LIN {X 0,Y 304.468,Z 656.126,A -85,B 0,C 180,E1 -16142.067,E2 -16142.067} C_VEL
LIN {X 0,Y 304.044,Z 658.272,A -85,B 0,C 180,E1 -16143.694,E2 -16143.694} C_VEL
LIN {X 0,Y 303.714,Z 660.484,A -85,B 0,C 180,E1 -16145.912,E2 -16145.912} C_VEL
LIN {X 0,Y 303.547,Z 662.089,A -85,B 0,C 180,E1 -16148.692,E2 -16148.692} C_VEL
LIN {X 0,Y 303.552,Z 662.479,A -85,B 0,C 180,E1 -16150.411,E2 -16150.411} C_VEL
LIN {X 0,Y 303.63,Z 662.376,A -85,B 0,C 180,E1 -16152.209,E2 -16152.209} C_VEL
LIN {X 0,Y 303.809,Z 661.626,A -85,B 0,C 180,E1 -16154.182,E2 -16154.182} C_VEL
LIN {X 0,Y 304.102,Z 660.328,A -85,B 0,C 180,E1 -16156.106,E2 -16156.106} C_VEL
LIN {X 0,Y 304.595,Z 658.473,A -85,B 0,C 180,E1 -16158,E2 -16158} C_VEL
LIN {X 0,Y 305.42,Z 654.743,A -85,B 0,C 180,E1 -16160.682,E2 -16160.682} C_VEL
LIN {X 0,Y 306.67,Z 649.557,A -85,B 0,C 180,E1 -16163.426,E2 -16163.426} C_VEL
LIN {X 0,Y 308.375,Z 642.973,A -85,B 0,C 180,E1 -16166.107,E2 -16166.107} C_VEL
LIN {X 0,Y 310.419,Z 635.217,A -85,B 0,C 180,E1 -16168.618,E2 -16168.618} C_VEL
LIN {X 0,Y 312.569,Z 627.022,A -85,B 0,C 180,E1 -16170.788,E2 -16170.788} C_VEL
LIN {X 0,Y 315.085,Z 617.352,A -85,B 0,C 180,E1 -16172.91,E2 -16172.91} C_VEL
LIN {X 0,Y 317.539,Z 607.207,A -85,B 0,C 180,E1 -16174.766,E2 -16174.766} C_VEL
LIN {X 0,Y 320.243,Z 595.361,A -85,B 0,C 180,E1 -16176.561,E2 -16176.561} C_VEL
LIN {X 0,Y 322.857,Z 582.894,A -85,B 0,C 180,E1 -16178.112,E2 -16178.112} C_VEL
LIN {X 0,Y 325.28,Z 569.513,A -85,B 0,C 180,E1 -16179.477,E2 -16179.477} C_VEL
LIN {X 0,Y 325.963,Z 565.676,A -85,B 0,C 180,E1 -16179.818,E2 -16179.818} C_VEL
LIN {X 0,Y 325.947,Z 562.448,A -85,B 0,C 180,E1 -16180.17,E2 -16180.17} C_VEL
LIN {X 0,Y 324.622,Z 558.931,A -85,B 0,C 180,E1 -16180.704,E2 -16180.704} C_VEL
LIN {X 0,Y 321.402,Z 554.854,A -85,B 0,C 180,E1 -16181.521,E2 -16181.521} C_VEL
LIN {X 0,Y 315.876,Z 549.196,A -85,B 0,C 180,E1 -16182.776,E2 -16182.776} C_VEL
LIN {X 0,Y 313.449,Z 544.969,A -85,B 0,C 180,E1 -16183.488,E2 -16183.488} C_VEL
LIN {X 0,Y 308.452,Z 533.574,A -85,B 0,C 180,E1 -16185.105,E2 -16185.105} C_VEL
LIN {X 0,Y 303.295,Z 523.807,A -85,B 0,C 180,E1 -16186.575,E2 -16186.575} C_VEL
LIN {X 0,Y 300.999,Z 519.913,A -85,B 0,C 180,E1 -16187.184,E2 -16187.184} C_VEL
LIN {X 0,Y 299.322,Z 517.279,A -85,B 0,C 180,E1 -16187.628,E2 -16187.628} C_VEL
LIN {X 0,Y 298.927,Z 515.725,A -85,B 0,C 180,E1 -16187.783,E2 -16187.783} C_VEL
LIN {X 0,Y 299.077,Z 513.977,A -85,B 0,C 180,E1 -16191.894,E2 -16191.894} C_VEL
LIN {X 0,Y 298.86,Z 513.035,A -85,B 0,C 180,E1 -16194.602,E2 -16194.602} C_VEL
LIN {X 0,Y 298.922,Z 511.875,A -85,B 0,C 180,E1 -16198.652,E2 -16198.652} C_VEL
LIN {X 0,Y 298.922,Z 511.874,A -85,B 0,C 180,E1 -16201.347,E2 -16201.347} C_VEL
LIN {X 0,Y 298.796,Z 511.89,A -85,B 0,C 180,E1 -16206.753,E2 -16206.753} C_VEL
LIN {X 0,Y 298.679,Z 511.903,A -85,B 0,C 180,E1 -16209.48,E2 -16209.48} C_VEL
LIN {X 0,Y 298.55,Z 511.918,A -85,B 0,C 180,E1 -16213.615,E2 -16213.615} C_VEL
LIN {X 0,Y 298.546,Z 511.923,A -85,B 0,C 180,E1 -16216.408,E2 -16216.408} C_VEL
LIN {X 0,Y 298.509,Z 511.924,A -85,B 0,C 180,E1 -16219.654,E2 -16219.654} C_VEL
LIN {X 0,Y 298.446,Z 512.07,A -85,B 0,C 180,E1 -16222.134,E2 -16222.134} C_VEL
LIN {X 0,Y 298.697,Z 513.171,A -85,B 0,C 180,E1 -16225.056,E2 -16225.056} C_VEL
LIN {X 0,Y 298.927,Z 514.632,A -85,B 0,C 180,E1 -16228.048,E2 -16228.048} C_VEL
LIN {X 0,Y 299.194,Z 516.442,A -85,B 0,C 180,E1 -16231.116,E2 -16231.116} C_VEL
LIN {X 0,Y 299.664,Z 519.004,A -85,B 0,C 180,E1 -16234.83,E2 -16234.83} C_VEL
LIN {X 0,Y 300.312,Z 522.622,A -85,B 0,C 180,E1 -16239.187,E2 -16239.187} C_VEL
LIN {X 0,Y 300.797,Z 525.954,A -85,B 0,C 180,E1 -16242.654,E2 -16242.654} C_VEL
LIN {X 0,Y 301.367,Z 529.88,A -85,B 0,C 180,E1 -16246.297,E2 -16246.297} C_VEL
LIN {X 0,Y 301.234,Z 532.28,A -85,B 0,C 180,E1 -16248.295,E2 -16248.295} C_VEL
LIN {X 0,Y 300.435,Z 537.264,A -85,B 0,C 180,E1 -16252.116,E2 -16252.116} C_VEL
LIN {X 0,Y 300.324,Z 537.751,A -85,B 0,C 180,E1 -16252.464,E2 -16252.464} C_VEL
LIN {X 0,Y 301.249,Z 540.977,A -85,B 0,C 180,E1 -16252.761,E2 -16252.761} C_VEL
LIN {X 0,Y 302.452,Z 543.428,A -85,B 0,C 180,E1 -16253.081,E2 -16253.081} C_VEL
LIN {X 0,Y 307.21,Z 556.096,A -85,B 0,C 180,E1 -16254.515,E2 -16254.515} C_VEL
LIN {X 0,Y 310.981,Z 569.368,A -85,B 0,C 180,E1 -16255.971,E2 -16255.971} C_VEL
LIN {X 0,Y 313.752,Z 583.061,A -85,B 0,C 180,E1 -16257.48,E2 -16257.48} C_VEL
LIN {X 0,Y 315.221,Z 596.358,A -85,B 0,C 180,E1 -16258.972,E2 -16258.972} C_VEL
LIN {X 0,Y 315.648,Z 607.148,A -85,B 0,C 180,E1 -16260.266,E2 -16260.266} C_VEL
LIN {X 0,Y 314.902,Z 611.825,A -85,B 0,C 180,E1 -16260.777,E2 -16260.777} C_VEL
LIN {X 0,Y 311.977,Z 624.765,A -85,B 0,C 180,E1 -16262.314,E2 -16262.314} C_VEL
LIN {X 0,Y 309.129,Z 636.736,A -85,B 0,C 180,E1 -16264.046,E2 -16264.046} C_VEL
LIN {X 0,Y 306.332,Z 647.818,A -85,B 0,C 180,E1 -16265.969,E2 -16265.969} C_VEL
LIN {X 0,Y 303.981,Z 657.256,A -85,B 0,C 180,E1 -16267.935,E2 -16267.935} C_VEL
LIN {X 0,Y 301.707,Z 666.564,A -85,B 0,C 180,E1 -16270.259,E2 -16270.259} C_VEL
LIN {X 0,Y 299.707,Z 675.414,A -85,B 0,C 180,E1 -16272.955,E2 -16272.955} C_VEL
LIN {X 0,Y 298.197,Z 682.598,A -85,B 0,C 180,E1 -16275.672,E2 -16275.672} C_VEL
LIN {X 0,Y 297.264,Z 688.305,A -85,B 0,C 180,E1 -16278.406,E2 -16278.406} C_VEL
LIN {X 0,Y 296.881,Z 691.721,A -85,B 0,C 180,E1 -16280.461,E2 -16280.461} C_VEL
LIN {X 0,Y 296.637,Z 695.166,A -85,B 0,C 180,E1 -16283.196,E2 -16283.196} C_VEL
LIN {X 0,Y 296.651,Z 697.347,A -85,B 0,C 180,E1 -16285.924,E2 -16285.924} C_VEL
LIN {X 0,Y 296.763,Z 698.349,A -85,B 0,C 180,E1 -16288.642,E2 -16288.642} C_VEL
LIN {X 0,Y 296.887,Z 698.412,A -85,B 0,C 180,E1 -16289.999,E2 -16289.999} C_VEL
LIN {X 0,Y 296.672,Z 697.618,A -85,B 0,C 180,E1 -16292.715,E2 -16292.715} C_VEL
LIN {X 0,Y 296.689,Z 695.633,A -85,B 0,C 180,E1 -16295.436,E2 -16295.436} C_VEL
LIN {X 0,Y 296.777,Z 692.368,A -85,B 0,C 180,E1 -16298.168,E2 -16298.168} C_VEL
LIN {X 0,Y 297.068,Z 687.756,A -85,B 0,C 180,E1 -16300.909,E2 -16300.909} C_VEL
LIN {X 0,Y 297.844,Z 681.725,A -85,B 0,C 180,E1 -16303.647,E2 -16303.647} C_VEL
LIN {X 0,Y 299.149,Z 674.123,A -85,B 0,C 180,E1 -16306.374,E2 -16306.374} C_VEL
LIN {X 0,Y 300.619,Z 665.958,A -85,B 0,C 180,E1 -16308.75,E2 -16308.75} C_VEL
LIN {X 0,Y 302.441,Z 657.688,A -85,B 0,C 180,E1 -16310.754,E2 -16310.754} C_VEL
LIN {X 0,Y 304.456,Z 647.468,A -85,B 0,C 180,E1 -16312.846,E2 -16312.846} C_VEL
LIN {X 0,Y 306.936,Z 635.389,A -85,B 0,C 180,E1 -16314.88,E2 -16314.88} C_VEL
LIN {X 0,Y 309.172,Z 623.827,A -85,B 0,C 180,E1 -16316.493,E2 -16316.493} C_VEL
LIN {X 0,Y 311.592,Z 611.493,A -85,B 0,C 180,E1 -16317.905,E2 -16317.905} C_VEL
LIN {X 0,Y 312.384,Z 605.5,A -85,B 0,C 180,E1 -16318.519,E2 -16318.519} C_VEL
LIN {X 0,Y 310.846,Z 591.329,A -85,B 0,C 180,E1 -16320.03,E2 -16320.03} C_VEL
LIN {X 0,Y 308.538,Z 577.479,A -85,B 0,C 180,E1 -16321.332,E2 -16321.332} C_VEL
LIN {X 0,Y 305.347,Z 563.007,A -85,B 0,C 180,E1 -16322.536,E2 -16322.536} C_VEL
LIN {X 0,Y 301.249,Z 548.178,A -85,B 0,C 180,E1 -16323.625,E2 -16323.625} C_VEL
LIN {X 0,Y 299.596,Z 542.829,A -85,B 0,C 180,E1 -16323.986,E2 -16323.986} C_VEL
LIN {X 0,Y 299.525,Z 541.899,A -85,B 0,C 180,E1 -16324.059,E2 -16324.059} C_VEL
LIN {X 0,Y 300.214,Z 536.845,A -85,B 0,C 180,E1 -16327.491,E2 -16327.491} C_VEL
LIN {X 0,Y 301.015,Z 532.092,A -85,B 0,C 180,E1 -16330.822,E2 -16330.822} C_VEL
LIN {X 0,Y 301.291,Z 529.646,A -85,B 0,C 180,E1 -16332.566,E2 -16332.566} C_VEL
LIN {X 0,Y 300.918,Z 525.827,A -85,B 0,C 180,E1 -16335.521,E2 -16335.521} C_VEL
LIN {X 0,Y 300.088,Z 521.552,A -85,B 0,C 180,E1 -16339.024,E2 -16339.024} C_VEL
LIN {X 0,Y 299.269,Z 517.042,A -85,B 0,C 180,E1 -16342.98,E2 -16342.98} C_VEL
LIN {X 0,Y 298.814,Z 514.18,A -85,B 0,C 180,E1 -16345.635,E2 -16345.635} C_VEL
LIN {X 0,Y 298.394,Z 511.938,A -85,B 0,C 180,E1 -16347.981,E2 -16347.981} C_VEL
LIN {X 0,Y 298.461,Z 511.933,A -85,B 0,C 180,E1 -16351.905,E2 -16351.905} C_VEL
LIN {X 0,Y 298.475,Z 511.93,A -85,B 0,C 180,E1 -16354.924,E2 -16354.924} C_VEL
LIN {X 0,Y 298.431,Z 511.938,A -85,B 0,C 180,E1 -16359.314,E2 -16359.314} C_VEL
LIN {X 0,Y 298.529,Z 511.923,A -85,B 0,C 180,E1 -16362.179,E2 -16362.179} C_VEL
LIN {X 0,Y 298.585,Z 511.916,A -85,B 0,C 180,E1 -16364.995,E2 -16364.995} C_VEL
LIN {X 0,Y 298.587,Z 511.914,A -85,B 0,C 180,E1 -16369.147,E2 -16369.147} C_VEL
LIN {X 0,Y 298.75,Z 511.891,A -85,B 0,C 180,E1 -16371.886,E2 -16371.886} C_VEL
LIN {X 0,Y 298.654,Z 511.905,A -85,B 0,C 180,E1 -16374.599,E2 -16374.599} C_VEL
LIN {X 0,Y 298.919,Z 511.869,A -85,B 0,C 180,E1 -16378.653,E2 -16378.653} C_VEL
LIN {X 0,Y 298.917,Z 511.865,A -85,B 0,C 180,E1 -16381.348,E2 -16381.348} C_VEL
LIN {X 0,Y 298.782,Z 511.89,A -85,B 0,C 180,E1 -16386.755,E2 -16386.755} C_VEL
LIN {X 0,Y 298.627,Z 511.908,A -85,B 0,C 180,E1 -16389.483,E2 -16389.483} C_VEL
LIN {X 0,Y 298.544,Z 511.913,A -85,B 0,C 180,E1 -16393.616,E2 -16393.616} C_VEL
LIN {X 0,Y 298.541,Z 511.919,A -85,B 0,C 180,E1 -16396.41,E2 -16396.41} C_VEL
LIN {X 0,Y 298.504,Z 511.926,A -85,B 0,C 180,E1 -16399.656,E2 -16399.656} C_VEL
LIN {X 0,Y 298.451,Z 511.922,A -85,B 0,C 180,E1 -16403.599,E2 -16403.599} C_VEL
LIN {X 0,Y 298.484,Z 511.922,A -85,B 0,C 180,E1 -16406.576,E2 -16406.576} C_VEL
LIN {X 0,Y 298.417,Z 511.94,A -85,B 0,C 180,E1 -16409.642,E2 -16409.642} C_VEL
LIN {X 0,Y 298.393,Z 511.936,A -85,B 0,C 180,E1 -16412.801,E2 -16412.801} C_VEL
LIN {X 0,Y 298.467,Z 511.92,A -85,B 0,C 180,E1 -16416.815,E2 -16416.815} C_VEL
LIN {X 0,Y 298.454,Z 511.933,A -85,B 0,C 180,E1 -16421.251,E2 -16421.251} C_VEL
LIN {X 0,Y 298.487,Z 511.923,A -85,B 0,C 180,E1 -16425.062,E2 -16425.062} C_VEL
LIN {X 0,Y 298.455,Z 511.929,A -85,B 0,C 180,E1 -16428.898,E2 -16428.898} C_VEL
LIN {X 0,Y 298.469,Z 511.931,A -85,B 0,C 180,E1 -16433.188,E2 -16433.188} C_VEL
LIN {X 0,Y 298.395,Z 511.936,A -85,B 0,C 180,E1 -16437.201,E2 -16437.201} C_VEL
LIN {X 0,Y 298.433,Z 511.935,A -85,B 0,C 180,E1 -16440.616,E2 -16440.616} C_VEL
LIN {X 0,Y 298.485,Z 511.925,A -85,B 0,C 180,E1 -16443.475,E2 -16443.475} C_VEL
LIN {X 0,Y 298.438,Z 511.933,A -85,B 0,C 180,E1 -16446.698,E2 -16446.698} C_VEL
LIN {X 0,Y 298.542,Z 511.916,A -85,B 0,C 180,E1 -16450.758,E2 -16450.758} C_VEL
LIN {X 0,Y 298.597,Z 511.912,A -85,B 0,C 180,E1 -16454.996,E2 -16454.996} C_VEL
LIN {X 0,Y 298.595,Z 511.915,A -85,B 0,C 180,E1 -16459.148,E2 -16459.148} C_VEL
LIN {X 0,Y 298.723,Z 511.901,A -85,B 0,C 180,E1 -16461.886,E2 -16461.886} C_VEL
LIN {X 0,Y 298.66,Z 511.903,A -85,B 0,C 180,E1 -16464.6,E2 -16464.6} C_VEL
LIN {X 0,Y 298.929,Z 511.872,A -85,B 0,C 180,E1 -16468.654,E2 -16468.654} C_VEL
LIN {X 0,Y 298.863,Z 511.881,A -85,B 0,C 180,E1 -16471.348,E2 -16471.348} C_VEL
LIN {X 0,Y 298.253,Z 512.084,A -85,B 0,C 180,E1 -16476.003,E2 -16476.003} C_VEL
LIN {X 0,Y 299.348,Z 515.022,A -85,B 0,C 180,E1 -16476.234,E2 -16476.234} C_VEL
LIN {X 0,Y 302.643,Z 522.4,A -85,B 0,C 180,E1 -16476.899,E2 -16476.899} C_VEL
LIN {X 0,Y 307.781,Z 536.221,A -85,B 0,C 180,E1 -16478.189,E2 -16478.189} C_VEL
LIN {X 0,Y 311.731,Z 548.462,A -85,B 0,C 180,E1 -16479.446,E2 -16479.446} C_VEL
LIN {X 0,Y 315.162,Z 561.803,A -85,B 0,C 180,E1 -16480.942,E2 -16480.942} C_VEL
LIN {X 0,Y 313.165,Z 576.214,A -85,B 0,C 180,E1 -16482.31,E2 -16482.31} C_VEL
LIN {X 0,Y 310.649,Z 590.58,A -85,B 0,C 180,E1 -16484.004,E2 -16484.004} C_VEL
LIN {X 0,Y 308.481,Z 602.271,A -85,B 0,C 180,E1 -16485.697,E2 -16485.697} C_VEL
LIN {X 0,Y 306.015,Z 613.873,A -85,B 0,C 180,E1 -16487.717,E2 -16487.717} C_VEL
LIN {X 0,Y 303.761,Z 624.438,A -85,B 0,C 180,E1 -16489.959,E2 -16489.959} C_VEL
LIN {X 0,Y 301.856,Z 633.291,A -85,B 0,C 180,E1 -16492.231,E2 -16492.231} C_VEL
LIN {X 0,Y 300.067,Z 641.854,A -85,B 0,C 180,E1 -16494.935,E2 -16494.935} C_VEL
LIN {X 0,Y 298.855,Z 648.075,A -85,B 0,C 180,E1 -16497.369,E2 -16497.369} C_VEL
LIN {X 0,Y 298.014,Z 652.821,A -85,B 0,C 180,E1 -16499.686,E2 -16499.686} C_VEL
LIN {X 0,Y 297.458,Z 656.235,A -85,B 0,C 180,E1 -16501.725,E2 -16501.725} C_VEL
LIN {X 0,Y 296.798,Z 659.814,A -85,B 0,C 180,E1 -16504.632,E2 -16504.632} C_VEL
LIN {X 0,Y 296.598,Z 661.257,A -85,B 0,C 180,E1 -16506.326,E2 -16506.326} C_VEL
LIN {X 0,Y 296.475,Z 662.439,A -85,B 0,C 180,E1 -16508.53,E2 -16508.53} C_VEL
LIN {X 0,Y 296.478,Z 662.939,A -85,B 0,C 180,E1 -16510.662,E2 -16510.662} C_VEL
LIN {X 0,Y 296.636,Z 662.495,A -85,B 0,C 180,E1 -16513.399,E2 -16513.399} C_VEL
LIN {X 0,Y 296.868,Z 661.589,A -85,B 0,C 180,E1 -16515.252,E2 -16515.252} C_VEL
LIN {X 0,Y 297.275,Z 660.07,A -85,B 0,C 180,E1 -16517.129,E2 -16517.129} C_VEL
LIN {X 0,Y 298.067,Z 657.03,A -85,B 0,C 180,E1 -16519.775,E2 -16519.775} C_VEL
LIN {X 0,Y 299.357,Z 651.736,A -85,B 0,C 180,E1 -16522.96,E2 -16522.96} C_VEL
LIN {X 0,Y 300.826,Z 646.331,A -85,B 0,C 180,E1 -16525.443,E2 -16525.443} C_VEL
LIN {X 0,Y 302.83,Z 639.188,A -85,B 0,C 180,E1 -16528.043,E2 -16528.043} C_VEL
LIN {X 0,Y 305.305,Z 630.25,A -85,B 0,C 180,E1 -16530.648,E2 -16530.648} C_VEL
LIN {X 0,Y 307.914,Z 620.784,A -85,B 0,C 180,E1 -16532.892,E2 -16532.892} C_VEL
LIN {X 0,Y 310.755,Z 609.932,A -85,B 0,C 180,E1 -16535.007,E2 -16535.007} C_VEL
LIN {X 0,Y 313.475,Z 598.769,A -85,B 0,C 180,E1 -16536.809,E2 -16536.809} C_VEL
LIN {X 0,Y 316.378,Z 585.853,A -85,B 0,C 180,E1 -16538.517,E2 -16538.517} C_VEL
LIN {X 0,Y 318.946,Z 572.612,A -85,B 0,C 180,E1 -16539.944,E2 -16539.944} C_VEL
LIN {X 0,Y 319.911,Z 567.296,A -85,B 0,C 180,E1 -16540.426,E2 -16540.426} C_VEL
LIN {X 0,Y 317.233,Z 556.251,A -85,B 0,C 180,E1 -16541.931,E2 -16541.931} C_VEL
LIN {X 0,Y 313.449,Z 544.969,A -85,B 0,C 180,E1 -16543.488,E2 -16543.488} C_VEL
LIN {X 0,Y 311.819,Z 542.414,A -85,B 0,C 180,E1 -16543.954,E2 -16543.954} C_VEL
LIN {X 0,Y 307.83,Z 539.626,A -85,B 0,C 180,E1 -16544.814,E2 -16544.814} C_VEL
LIN {X 0,Y 303.71,Z 536.917,A -85,B 0,C 180,E1 -16545.693,E2 -16545.693} C_VEL
LIN {X 0,Y 301.871,Z 534.458,A -85,B 0,C 180,E1 -16546.182,E2 -16546.182} C_VEL
LIN {X 0,Y 298.564,Z 528.116,A -85,B 0,C 180,E1 -16547.207,E2 -16547.207} C_VEL
LIN {X 0,Y 296.802,Z 524.957,A -85,B 0,C 180,E1 -16547.738,E2 -16547.738} C_VEL
LIN {X 0,Y 294.822,Z 521.445,A -85,B 0,C 180,E1 -16548.31,E2 -16548.31} C_VEL
LIN {X 0,Y 292.662,Z 518.54,A -85,B 0,C 180,E1 -16548.894,E2 -16548.894} C_VEL
LIN {X 0,Y 291.963,Z 516.396,A -85,B 0,C 180,E1 -16549.16,E2 -16549.16} C_VEL
LIN {X 0,Y 292.098,Z 515.364,A -85,B 0,C 180,E1 -16551.699,E2 -16551.699} C_VEL
LIN {X 0,Y 291.915,Z 514.421,A -85,B 0,C 180,E1 -16554.473,E2 -16554.473} C_VEL
LIN {X 0,Y 291.946,Z 513.188,A -85,B 0,C 180,E1 -16558.62,E2 -16558.62} C_VEL
LIN {X 0,Y 291.888,Z 512.75,A -85,B 0,C 180,E1 -16561.379,E2 -16561.379} C_VEL
LIN {X 0,Y 291.745,Z 512.767,A -85,B 0,C 180,E1 -16566.917,E2 -16566.917} C_VEL
LIN {X 0,Y 291.628,Z 512.781,A -85,B 0,C 180,E1 -16569.711,E2 -16569.711} C_VEL
LIN {X 0,Y 291.52,Z 512.795,A -85,B 0,C 180,E1 -16573.95,E2 -16573.95} C_VEL
LIN {X 0,Y 291.485,Z 512.8,A -85,B 0,C 180,E1 -16576.817,E2 -16576.817} C_VEL
LIN {X 0,Y 291.482,Z 512.993,A -85,B 0,C 180,E1 -16579.892,E2 -16579.892} C_VEL
LIN {X 0,Y 291.676,Z 514.441,A -85,B 0,C 180,E1 -16584.18,E2 -16584.18} C_VEL
LIN {X 0,Y 291.943,Z 515.792,A -85,B 0,C 180,E1 -16587.218,E2 -16587.218} C_VEL
LIN {X 0,Y 292.188,Z 517.522,A -85,B 0,C 180,E1 -16590.338,E2 -16590.338} C_VEL
LIN {X 0,Y 292.534,Z 519.609,A -85,B 0,C 180,E1 -16593.543,E2 -16593.543} C_VEL
LIN {X 0,Y 292.983,Z 522.099,A -85,B 0,C 180,E1 -16596.847,E2 -16596.847} C_VEL
LIN {X 0,Y 293.498,Z 525.046,A -85,B 0,C 180,E1 -16600.28,E2 -16600.28} C_VEL
LIN {X 0,Y 294.068,Z 528.9,A -85,B 0,C 180,E1 -16604.195,E2 -16604.195} C_VEL
LIN {X 0,Y 294.367,Z 531.02,A -85,B 0,C 180,E1 -16606.182,E2 -16606.182} C_VEL
LIN {X 0,Y 294.101,Z 534.266,A -85,B 0,C 180,E1 -16608.917,E2 -16608.917} C_VEL
LIN {X 0,Y 293.625,Z 537.124,A -85,B 0,C 180,E1 -16611.157,E2 -16611.157} C_VEL
LIN {X 0,Y 294.568,Z 540.375,A -85,B 0,C 180,E1 -16611.483,E2 -16611.483} C_VEL
LIN {X 0,Y 295.873,Z 543.008,A -85,B 0,C 180,E1 -16611.86,E2 -16611.86} C_VEL
LIN {X 0,Y 301.07,Z 556.672,A -85,B 0,C 180,E1 -16613.538,E2 -16613.538} C_VEL
LIN {X 0,Y 304.668,Z 569.174,A -85,B 0,C 180,E1 -16615.01,E2 -16615.01} C_VEL
LIN {X 0,Y 307.4,Z 582.594,A -85,B 0,C 180,E1 -16616.563,E2 -16616.563} C_VEL
LIN {X 0,Y 308.824,Z 594.993,A -85,B 0,C 180,E1 -16618.015,E2 -16618.015} C_VEL
LIN {X 0,Y 309.388,Z 608.259,A -85,B 0,C 180,E1 -16619.677,E2 -16619.677} C_VEL
LIN {X 0,Y 308.086,Z 615.217,A -85,B 0,C 180,E1 -16620.468,E2 -16620.468} C_VEL
LIN {X 0,Y 304.882,Z 628.503,A -85,B 0,C 180,E1 -16622.173,E2 -16622.173} C_VEL
LIN {X 0,Y 301.721,Z 640.753,A -85,B 0,C 180,E1 -16624.103,E2 -16624.103} C_VEL
LIN {X 0,Y 298.552,Z 652.667,A -85,B 0,C 180,E1 -16626.41,E2 -16626.41} C_VEL
LIN {X 0,Y 296.015,Z 662.664,A -85,B 0,C 180,E1 -16628.773,E2 -16628.773} C_VEL
LIN {X 0,Y 293.793,Z 671.055,A -85,B 0,C 180,E1 -16631.159,E2 -16631.159} C_VEL
LIN {X 0,Y 291.966,Z 678.98,A -85,B 0,C 180,E1 -16633.929,E2 -16633.929} C_VEL
LIN {X 0,Y 290.691,Z 685.343,A -85,B 0,C 180,E1 -16636.721,E2 -16636.721} C_VEL
LIN {X 0,Y 289.91,Z 690.326,A -85,B 0,C 180,E1 -16639.524,E2 -16639.524} C_VEL
LIN {X 0,Y 289.634,Z 693.242,A -85,B 0,C 180,E1 -16641.628,E2 -16641.628} C_VEL
LIN {X 0,Y 289.554,Z 696.035,A -85,B 0,C 180,E1 -16644.428,E2 -16644.428} C_VEL
LIN {X 0,Y 289.587,Z 697.586,A -85,B 0,C 180,E1 -16647.217,E2 -16647.217} C_VEL
LIN {X 0,Y 289.798,Z 697.972,A -85,B 0,C 180,E1 -16649.999,E2 -16649.999} C_VEL
LIN {X 0,Y 289.595,Z 697.146,A -85,B 0,C 180,E1 -16652.781,E2 -16652.781} C_VEL
LIN {X 0,Y 289.622,Z 695.126,A -85,B 0,C 180,E1 -16655.569,E2 -16655.569} C_VEL
LIN {X 0,Y 289.699,Z 691.837,A -85,B 0,C 180,E1 -16658.369,E2 -16658.369} C_VEL
LIN {X 0,Y 290.028,Z 687.187,A -85,B 0,C 180,E1 -16661.177,E2 -16661.177} C_VEL
LIN {X 0,Y 290.866,Z 681.11,A -85,B 0,C 180,E1 -16663.981,E2 -16663.981} C_VEL
LIN {X 0,Y 292.251,Z 673.454,A -85,B 0,C 180,E1 -16666.772,E2 -16666.772} C_VEL
LIN {X 0,Y 293.825,Z 665.23,A -85,B 0,C 180,E1 -16669.2,E2 -16669.2} C_VEL
LIN {X 0,Y 295.673,Z 656.884,A -85,B 0,C 180,E1 -16671.252,E2 -16671.252} C_VEL
LIN {X 0,Y 297.78,Z 646.834,A -85,B 0,C 180,E1 -16673.338,E2 -16673.338} C_VEL
LIN {X 0,Y 300.4,Z 634.412,A -85,B 0,C 180,E1 -16675.459,E2 -16675.459} C_VEL
LIN {X 0,Y 303.074,Z 621.461,A -85,B 0,C 180,E1 -16677.256,E2 -16677.256} C_VEL
LIN {X 0,Y 305.564,Z 608.497,A -85,B 0,C 180,E1 -16678.716,E2 -16678.716} C_VEL
LIN {X 0,Y 305.611,Z 605.241,A -85,B 0,C 180,E1 -16679.089,E2 -16679.089} C_VEL
LIN {X 0,Y 304.02,Z 590.859,A -85,B 0,C 180,E1 -16680.673,E2 -16680.673} C_VEL
LIN {X 0,Y 301.593,Z 576.374,A -85,B 0,C 180,E1 -16682.077,E2 -16682.077} C_VEL
LIN {X 0,Y 298.299,Z 561.765,A -85,B 0,C 180,E1 -16683.324,E2 -16683.324} C_VEL
LIN {X 0,Y 294.285,Z 547.64,A -85,B 0,C 180,E1 -16684.395,E2 -16684.395} C_VEL
LIN {X 0,Y 292.687,Z 542.207,A -85,B 0,C 180,E1 -16684.77,E2 -16684.77} C_VEL
LIN {X 0,Y 292.652,Z 541.489,A -85,B 0,C 180,E1 -16684.855,E2 -16684.855} C_VEL
LIN {X 0,Y 293.586,Z 535.209,A -85,B 0,C 180,E1 -16689.276,E2 -16689.276} C_VEL
LIN {X 0,Y 294.19,Z 531.145,A -85,B 0,C 180,E1 -16692.221,E2 -16692.221} C_VEL
LIN {X 0,Y 294.167,Z 528.562,A -85,B 0,C 180,E1 -16694.215,E2 -16694.215} C_VEL
LIN {X 0,Y 293.344,Z 523.995,A -85,B 0,C 180,E1 -16697.96,E2 -16697.96} C_VEL
LIN {X 0,Y 292.383,Z 518.868,A -85,B 0,C 180,E1 -16702.485,E2 -16702.485} C_VEL
LIN {X 0,Y 291.71,Z 514.79,A -85,B 0,C 180,E1 -16706.35,E2 -16706.35} C_VEL
LIN {X 0,Y 291.341,Z 512.817,A -85,B 0,C 180,E1 -16708.354,E2 -16708.354} C_VEL
LIN {X 0,Y 291.379,Z 512.815,A -85,B 0,C 180,E1 -16711.159,E2 -16711.159} C_VEL
LIN {X 0,Y 291.408,Z 512.81,A -85,B 0,C 180,E1 -16714.272,E2 -16714.272} C_VEL
LIN {X 0,Y 291.366,Z 512.818,A -85,B 0,C 180,E1 -16717.299,E2 -16717.299} C_VEL
LIN {X 0,Y 291.45,Z 512.805,A -85,B 0,C 180,E1 -16720.27,E2 -16720.27} C_VEL
LIN {X 0,Y 291.547,Z 512.791,A -85,B 0,C 180,E1 -16724.624,E2 -16724.624} C_VEL
LIN {X 0,Y 291.53,Z 512.791,A -85,B 0,C 180,E1 -16728.881,E2 -16728.881} C_VEL
LIN {X 0,Y 291.7,Z 512.767,A -85,B 0,C 180,E1 -16731.689,E2 -16731.689} C_VEL
LIN {X 0,Y 291.624,Z 512.781,A -85,B 0,C 180,E1 -16734.469,E2 -16734.469} C_VEL
LIN {X 0,Y 291.885,Z 512.745,A -85,B 0,C 180,E1 -16738.621,E2 -16738.621} C_VEL
LIN {X 0,Y 291.883,Z 512.739,A -85,B 0,C 180,E1 -16741.38,E2 -16741.38} C_VEL
LIN {X 0,Y 291.73,Z 512.769,A -85,B 0,C 180,E1 -16746.919,E2 -16746.919} C_VEL
LIN {X 0,Y 291.567,Z 512.784,A -85,B 0,C 180,E1 -16749.715,E2 -16749.715} C_VEL
LIN {X 0,Y 291.514,Z 512.791,A -85,B 0,C 180,E1 -16753.951,E2 -16753.951} C_VEL
LIN {X 0,Y 291.48,Z 512.798,A -85,B 0,C 180,E1 -16756.819,E2 -16756.819} C_VEL
LIN {X 0,Y 291.444,Z 512.803,A -85,B 0,C 180,E1 -16759.876,E2 -16759.876} C_VEL
LIN {X 0,Y 291.394,Z 512.797,A -85,B 0,C 180,E1 -16764.206,E2 -16764.206} C_VEL
LIN {X 0,Y 291.417,Z 512.805,A -85,B 0,C 180,E1 -16767.273,E2 -16767.273} C_VEL
LIN {X 0,Y 291.334,Z 512.817,A -85,B 0,C 180,E1 -16770.438,E2 -16770.438} C_VEL
LIN {X 0,Y 291.341,Z 512.811,A -85,B 0,C 180,E1 -16773.7,E2 -16773.7} C_VEL
LIN {X 0,Y 291.401,Z 512.802,A -85,B 0,C 180,E1 -16777.263,E2 -16777.263} C_VEL
LIN {X 0,Y 291.403,Z 512.809,A -85,B 0,C 180,E1 -16780.632,E2 -16780.632} C_VEL
LIN {X 0,Y 291.404,Z 512.804,A -85,B 0,C 180,E1 -16784.381,E2 -16784.381} C_VEL
LIN {X 0,Y 291.389,Z 512.809,A -85,B 0,C 180,E1 -16788.391,E2 -16788.391} C_VEL
LIN {X 0,Y 291.387,Z 512.814,A -85,B 0,C 180,E1 -16791.166,E2 -16791.166} C_VEL
LIN {X 0,Y 291.385,Z 512.806,A -85,B 0,C 180,E1 -16794.631,E2 -16794.631} C_VEL
LIN {X 0,Y 291.372,Z 512.817,A -85,B 0,C 180,E1 -16797.952,E2 -16797.952} C_VEL
LIN {X 0,Y 291.384,Z 512.815,A -85,B 0,C 180,E1 -16801.16,E2 -16801.16} C_VEL
LIN {X 0,Y 291.419,Z 512.805,A -85,B 0,C 180,E1 -16804.273,E2 -16804.273} C_VEL
LIN {X 0,Y 291.384,Z 512.815,A -85,B 0,C 180,E1 -16807.301,E2 -16807.301} C_VEL
LIN {X 0,Y 291.461,Z 512.798,A -85,B 0,C 180,E1 -16810.271,E2 -16810.271} C_VEL
LIN {X 0,Y 291.558,Z 512.788,A -85,B 0,C 180,E1 -16814.625,E2 -16814.625} C_VEL
LIN {X 0,Y 291.539,Z 512.793,A -85,B 0,C 180,E1 -16818.882,E2 -16818.882} C_VEL
LIN {X 0,Y 291.672,Z 512.779,A -85,B 0,C 180,E1 -16821.688,E2 -16821.688} C_VEL
LIN {X 0,Y 291.63,Z 512.779,A -85,B 0,C 180,E1 -16824.469,E2 -16824.469} C_VEL
LIN {X 0,Y 291.895,Z 512.749,A -85,B 0,C 180,E1 -16828.621,E2 -16828.621} C_VEL
LIN {X 0,Y 291.821,Z 512.758,A -85,B 0,C 180,E1 -16831.381,E2 -16831.381} C_VEL
LIN {X 0,Y 291.287,Z 512.827,A -85,B 0,C 180,E1 -16835.192,E2 -16835.192} C_VEL
LIN {X 0,Y 292.436,Z 515.906,A -85,B 0,C 180,E1 -16835.474,E2 -16835.474} C_VEL
LIN {X 0,Y 296.593,Z 524.963,A -85,B 0,C 180,E1 -16836.35,E2 -16836.35} C_VEL
LIN {X 0,Y 301.963,Z 539.695,A -85,B 0,C 180,E1 -16837.805,E2 -16837.805} C_VEL
LIN {X 0,Y 306.01,Z 552.987,A -85,B 0,C 180,E1 -16839.252,E2 -16839.252} C_VEL
LIN {X 0,Y 308.645,Z 563.578,A -85,B 0,C 180,E1 -16840.496,E2 -16840.496} C_VEL
LIN {X 0,Y 306.493,Z 577.904,A -85,B 0,C 180,E1 -16841.91,E2 -16841.91} C_VEL
LIN {X 0,Y 304.021,Z 591.48,A -85,B 0,C 180,E1 -16843.565,E2 -16843.565} C_VEL
LIN {X 0,Y 301.688,Z 603.538,A -85,B 0,C 180,E1 -16845.367,E2 -16845.367} C_VEL
LIN {X 0,Y 299.182,Z 614.827,A -85,B 0,C 180,E1 -16847.393,E2 -16847.393} C_VEL
LIN {X 0,Y 296.82,Z 625.448,A -85,B 0,C 180,E1 -16849.719,E2 -16849.719} C_VEL
LIN {X 0,Y 294.897,Z 634.171,A -85,B 0,C 180,E1 -16852.033,E2 -16852.033} C_VEL
LIN {X 0,Y 293.273,Z 641.566,A -85,B 0,C 180,E1 -16854.405,E2 -16854.405} C_VEL
LIN {X 0,Y 291.83,Z 648.685,A -85,B 0,C 180,E1 -16857.23,E2 -16857.23} C_VEL
LIN {X 0,Y 290.969,Z 653.375,A -85,B 0,C 180,E1 -16859.594,E2 -16859.594} C_VEL
LIN {X 0,Y 290.263,Z 657.428,A -85,B 0,C 180,E1 -16862.187,E2 -16862.187} C_VEL
LIN {X 0,Y 289.747,Z 660.088,A -85,B 0,C 180,E1 -16864.442,E2 -16864.442} C_VEL
LIN {X 0,Y 289.414,Z 662.336,A -85,B 0,C 180,E1 -16867.379,E2 -16867.379} C_VEL
LIN {X 0,Y 289.369,Z 663.098,A -85,B 0,C 180,E1 -16869.159,E2 -16869.159} C_VEL
LIN {X 0,Y 289.393,Z 663.362,A -85,B 0,C 180,E1 -16871.162,E2 -16871.162} C_VEL
LIN {X 0,Y 289.534,Z 663.022,A -85,B 0,C 180,E1 -16873.263,E2 -16873.263} C_VEL
LIN {X 0,Y 289.816,Z 662.112,A -85,B 0,C 180,E1 -16875.311,E2 -16875.311} C_VEL
LIN {X 0,Y 290.603,Z 659.346,A -85,B 0,C 180,E1 -16878.565,E2 -16878.565} C_VEL
LIN {X 0,Y 291.483,Z 655.913,A -85,B 0,C 180,E1 -16881.178,E2 -16881.178} C_VEL
LIN {X 0,Y 292.786,Z 651.167,A -85,B 0,C 180,E1 -16883.883,E2 -16883.883} C_VEL
LIN {X 0,Y 294.686,Z 644.68,A -85,B 0,C 180,E1 -16886.733,E2 -16886.733} C_VEL
LIN {X 0,Y 296.655,Z 638.066,A -85,B 0,C 180,E1 -16889.056,E2 -16889.056} C_VEL
LIN {X 0,Y 298.964,Z 630.15,A -85,B 0,C 180,E1 -16891.358,E2 -16891.358} C_VEL
LIN {X 0,Y 301.906,Z 620.089,A -85,B 0,C 180,E1 -16893.749,E2 -16893.749} C_VEL
LIN {X 0,Y 304.714,Z 609.732,A -85,B 0,C 180,E1 -16895.78,E2 -16895.78} C_VEL
LIN {X 0,Y 307.713,Z 597.917,A -85,B 0,C 180,E1 -16897.684,E2 -16897.684} C_VEL
LIN {X 0,Y 310.543,Z 585.776,A -85,B 0,C 180,E1 -16899.291,E2 -16899.291} C_VEL
LIN {X 0,Y 313.202,Z 572.708,A -85,B 0,C 180,E1 -16900.71,E2 -16900.71} C_VEL
LIN {X 0,Y 313.865,Z 569.041,A -85,B 0,C 180,E1 -16901.052,E2 -16901.052} C_VEL
LIN {X 0,Y 310.972,Z 557.402,A -85,B 0,C 180,E1 -16902.744,E2 -16902.744} C_VEL
LIN {X 0,Y 306.71,Z 545.109,A -85,B 0,C 180,E1 -16904.551,E2 -16904.551} C_VEL
LIN {X 0,Y 302.363,Z 535.427,A -85,B 0,C 180,E1 -16906.028,E2 -16906.028} C_VEL
LIN {X 0,Y 301.871,Z 534.458,A -85,B 0,C 180,E1 -16906.182,E2 -16906.182} C_VEL
LIN {X 0,Y 300.078,Z 532.093,A -85,B 0,C 180,E1 -16906.678,E2 -16906.678} C_VEL
LIN {X 0,Y 296.01,Z 529.772,A -85,B 0,C 180,E1 -16907.601,E2 -16907.601} C_VEL
LIN {X 0,Y 291.855,Z 527.641,A -85,B 0,C 180,E1 -16908.568,E2 -16908.568} C_VEL
LIN {X 0,Y 289.881,Z 525.534,A -85,B 0,C 180,E1 -16909.122,E2 -16909.122} C_VEL
LIN {X 0,Y 287.582,Z 521.666,A -85,B 0,C 180,E1 -16909.838,E2 -16909.838} C_VEL
LIN {X 0,Y 285.756,Z 519.17,A -85,B 0,C 180,E1 -16910.385,E2 -16910.385} C_VEL
LIN {X 0,Y 285.111,Z 517.075,A -85,B 0,C 180,E1 -16910.661,E2 -16910.661} C_VEL
LIN {X 0,Y 284.963,Z 515.824,A -85,B 0,C 180,E1 -16914.338,E2 -16914.338} C_VEL
LIN {X 0,Y 285.012,Z 514.62,A -85,B 0,C 180,E1 -16918.586,E2 -16918.586} C_VEL
LIN {X 0,Y 284.911,Z 514.002,A -85,B 0,C 180,E1 -16921.413,E2 -16921.413} C_VEL
LIN {X 0,Y 284.6,Z 513.657,A -85,B 0,C 180,E1 -16925.668,E2 -16925.668} C_VEL
LIN {X 0,Y 284.665,Z 513.648,A -85,B 0,C 180,E1 -16929.054,E2 -16929.054} C_VEL
LIN {X 0,Y 284.474,Z 513.672,A -85,B 0,C 180,E1 -16932.846,E2 -16932.846} C_VEL
LIN {X 0,Y 284.48,Z 513.723,A -85,B 0,C 180,E1 -16935.768,E2 -16935.768} C_VEL
LIN {X 0,Y 284.557,Z 514.716,A -85,B 0,C 180,E1 -16940.228,E2 -16940.228} C_VEL
LIN {X 0,Y 284.808,Z 516.307,A -85,B 0,C 180,E1 -16944.802,E2 -16944.802} C_VEL
LIN {X 0,Y 285.062,Z 517.768,A -85,B 0,C 180,E1 -16947.932,E2 -16947.932} C_VEL
LIN {X 0,Y 285.323,Z 519.595,A -85,B 0,C 180,E1 -16951.149,E2 -16951.149} C_VEL
LIN {X 0,Y 285.709,Z 521.788,A -85,B 0,C 180,E1 -16954.455,E2 -16954.455} C_VEL
LIN {X 0,Y 286.272,Z 524.687,A -85,B 0,C 180,E1 -16958.224,E2 -16958.224} C_VEL
LIN {X 0,Y 286.683,Z 527.544,A -85,B 0,C 180,E1 -16961.445,E2 -16961.445} C_VEL
LIN {X 0,Y 287.243,Z 531.26,A -85,B 0,C 180,E1 -16965.197,E2 -16965.197} C_VEL
LIN {X 0,Y 287.338,Z 533.439,A -85,B 0,C 180,E1 -16967.203,E2 -16967.203} C_VEL
LIN {X 0,Y 286.914,Z 536.535,A -85,B 0,C 180,E1 -16969.733,E2 -16969.733} C_VEL
LIN {X 0,Y 287.898,Z 539.817,A -85,B 0,C 180,E1 -16970.1,E2 -16970.1} C_VEL
LIN {X 0,Y 289.262,Z 542.426,A -85,B 0,C 180,E1 -16970.525,E2 -16970.525} C_VEL
LIN {X 0,Y 293.446,Z 553.012,A -85,B 0,C 180,E1 -16971.941,E2 -16971.941} C_VEL
LIN {X 0,Y 297.246,Z 564.523,A -85,B 0,C 180,E1 -16973.431,E2 -16973.431} C_VEL
LIN {X 0,Y 300.259,Z 577.357,A -85,B 0,C 180,E1 -16975.007,E2 -16975.007} C_VEL
LIN {X 0,Y 302.276,Z 590.729,A -85,B 0,C 180,E1 -16976.661,E2 -16976.661} C_VEL
LIN {X 0,Y 303.098,Z 604.529,A -85,B 0,C 180,E1 -16978.416,E2 -16978.416} C_VEL
LIN {X 0,Y 302.945,Z 611.298,A -85,B 0,C 180,E1 -16979.311,E2 -16979.311} C_VEL
LIN {X 0,Y 299.492,Z 625.273,A -85,B 0,C 180,E1 -16981.053,E2 -16981.053} C_VEL
LIN {X 0,Y 296.409,Z 636.996,A -85,B 0,C 180,E1 -16982.843,E2 -16982.843} C_VEL
LIN {X 0,Y 293.34,Z 647.849,A -85,B 0,C 180,E1 -16984.832,E2 -16984.832} C_VEL
LIN {X 0,Y 290.362,Z 658.512,A -85,B 0,C 180,E1 -16987.215,E2 -16987.215} C_VEL
LIN {X 0,Y 287.928,Z 667.471,A -85,B 0,C 180,E1 -16989.645,E2 -16989.645} C_VEL
LIN {X 0,Y 286.01,Z 675.03,A -85,B 0,C 180,E1 -16992.112,E2 -16992.112} C_VEL
LIN {X 0,Y 284.229,Z 682.348,A -85,B 0,C 180,E1 -16995.068,E2 -16995.068} C_VEL
LIN {X 0,Y 283.238,Z 687.717,A -85,B 0,C 180,E1 -16997.824,E2 -16997.824} C_VEL
LIN {X 0,Y 282.741,Z 691.043,A -85,B 0,C 180,E1 -16999.979,E2 -16999.979} C_VEL
LIN {X 0,Y 282.469,Z 694.424,A -85,B 0,C 180,E1 -17002.853,E2 -17002.853} C_VEL
LIN {X 0,Y 282.481,Z 696.57,A -85,B 0,C 180,E1 -17005.719,E2 -17005.719} C_VEL
LIN {X 0,Y 282.577,Z 697.502,A -85,B 0,C 180,E1 -17008.574,E2 -17008.574} C_VEL
LIN {X 0,Y 282.709,Z 697.531,A -85,B 0,C 180,E1 -17009.999,E2 -17009.999} C_VEL
LIN {X 0,Y 282.52,Z 696.669,A -85,B 0,C 180,E1 -17012.851,E2 -17012.851} C_VEL
LIN {X 0,Y 282.599,Z 694.449,A -85,B 0,C 180,E1 -17015.869,E2 -17015.869} C_VEL
LIN {X 0,Y 282.62,Z 691.285,A -85,B 0,C 180,E1 -17018.58,E2 -17018.58} C_VEL
LIN {X 0,Y 282.994,Z 686.604,A -85,B 0,C 180,E1 -17021.459,E2 -17021.459} C_VEL
LIN {X 0,Y 283.898,Z 680.478,A -85,B 0,C 180,E1 -17024.332,E2 -17024.332} C_VEL
LIN {X 0,Y 285.345,Z 672.767,A -85,B 0,C 180,E1 -17027.19,E2 -17027.19} C_VEL
LIN {X 0,Y 287.053,Z 664.49,A -85,B 0,C 180,E1 -17029.671,E2 -17029.671} C_VEL
LIN {X 0,Y 289.371,Z 654.578,A -85,B 0,C 180,E1 -17032.113,E2 -17032.113} C_VEL
LIN {X 0,Y 291.511,Z 644.406,A -85,B 0,C 180,E1 -17034.194,E2 -17034.194} C_VEL
LIN {X 0,Y 293.977,Z 633.448,A -85,B 0,C 180,E1 -17036.057,E2 -17036.057} C_VEL
LIN {X 0,Y 296.442,Z 621.67,A -85,B 0,C 180,E1 -17037.726,E2 -17037.726} C_VEL
LIN {X 0,Y 298.905,Z 609.253,A -85,B 0,C 180,E1 -17039.174,E2 -17039.174} C_VEL
LIN {X 0,Y 298.795,Z 604.274,A -85,B 0,C 180,E1 -17039.773,E2 -17039.773} C_VEL
LIN {X 0,Y 297.244,Z 590.411,A -85,B 0,C 180,E1 -17041.342,E2 -17041.342} C_VEL
LIN {X 0,Y 294.758,Z 575.703,A -85,B 0,C 180,E1 -17042.803,E2 -17042.803} C_VEL
LIN {X 0,Y 291.074,Z 559.7,A -85,B 0,C 180,E1 -17044.211,E2 -17044.211} C_VEL
LIN {X 0,Y 286.447,Z 544.108,A -85,B 0,C 180,E1 -17045.431,E2 -17045.431} C_VEL
LIN {X 0,Y 285.712,Z 541.141,A -85,B 0,C 180,E1 -17045.644,E2 -17045.644} C_VEL
LIN {X 0,Y 286.61,Z 535.621,A -85,B 0,C 180,E1 -17049.607,E2 -17049.607} C_VEL
LIN {X 0,Y 287.212,Z 531.425,A -85,B 0,C 180,E1 -17052.77,E2 -17052.77} C_VEL
LIN {X 0,Y 286.963,Z 528.339,A -85,B 0,C 180,E1 -17055.252,E2 -17055.252} C_VEL
LIN {X 0,Y 286.207,Z 524.565,A -85,B 0,C 180,E1 -17058.471,E2 -17058.471} C_VEL
LIN {X 0,Y 285.486,Z 520.62,A -85,B 0,C 180,E1 -17062.017,E2 -17062.017} C_VEL
LIN {X 0,Y 284.878,Z 517.047,A -85,B 0,C 180,E1 -17065.43,E2 -17065.43} C_VEL
LIN {X 0,Y 284.313,Z 513.693,A -85,B 0,C 180,E1 -17069.056,E2 -17069.056} C_VEL
LIN {X 0,Y 284.39,Z 513.685,A -85,B 0,C 180,E1 -17072.826,E2 -17072.826} C_VEL
LIN {X 0,Y 284.325,Z 513.693,A -85,B 0,C 180,E1 -17076.704,E2 -17076.704} C_VEL
LIN {X 0,Y 284.395,Z 513.686,A -85,B 0,C 180,E1 -17081.262,E2 -17081.262} C_VEL
LIN {X 0,Y 284.484,Z 513.671,A -85,B 0,C 180,E1 -17084.459,E2 -17084.459} C_VEL
LIN {X 0,Y 284.481,Z 513.668,A -85,B 0,C 180,E1 -17088.602,E2 -17088.602} C_VEL
LIN {X 0,Y 284.65,Z 513.642,A -85,B 0,C 180,E1 -17091.481,E2 -17091.481} C_VEL
LIN {X 0,Y 284.595,Z 513.657,A -85,B 0,C 180,E1 -17094.332,E2 -17094.332} C_VEL
LIN {X 0,Y 284.851,Z 513.621,A -85,B 0,C 180,E1 -17098.587,E2 -17098.587} C_VEL
LIN {X 0,Y 284.849,Z 513.614,A -85,B 0,C 180,E1 -17101.414,E2 -17101.414} C_VEL
LIN {X 0,Y 284.681,Z 513.648,A -85,B 0,C 180,E1 -17107.091,E2 -17107.091} C_VEL
LIN {X 0,Y 284.511,Z 513.661,A -85,B 0,C 180,E1 -17109.958,E2 -17109.958} C_VEL
LIN {X 0,Y 284.47,Z 513.666,A -85,B 0,C 180,E1 -17114.304,E2 -17114.304} C_VEL
LIN {X 0,Y 284.418,Z 513.68,A -85,B 0,C 180,E1 -17117.249,E2 -17117.249} C_VEL
LIN {X 0,Y 284.372,Z 513.682,A -85,B 0,C 180,E1 -17120.243,E2 -17120.243} C_VEL
LIN {X 0,Y 284.363,Z 513.672,A -85,B 0,C 180,E1 -17123.876,E2 -17123.876} C_VEL
LIN {X 0,Y 284.392,Z 513.679,A -85,B 0,C 180,E1 -17127.175,E2 -17127.175} C_VEL
LIN {X 0,Y 284.293,Z 513.697,A -85,B 0,C 180,E1 -17131.275,E2 -17131.275} C_VEL
LIN {X 0,Y 284.358,Z 513.675,A -85,B 0,C 180,E1 -17135.356,E2 -17135.356} C_VEL
LIN {X 0,Y 284.334,Z 513.687,A -85,B 0,C 180,E1 -17138.166,E2 -17138.166} C_VEL
LIN {X 0,Y 284.342,Z 513.689,A -85,B 0,C 180,E1 -17142.143,E2 -17142.143} C_VEL
LIN {X 0,Y 284.351,Z 513.677,A -85,B 0,C 180,E1 -17146.21,E2 -17146.21} C_VEL
LIN {X 0,Y 284.35,Z 513.691,A -85,B 0,C 180,E1 -17150.015,E2 -17150.015} C_VEL
LIN {X 0,Y 284.355,Z 513.687,A -85,B 0,C 180,E1 -17153.619,E2 -17153.619} C_VEL
LIN {X 0,Y 284.308,Z 513.69,A -85,B 0,C 180,E1 -17157.191,E2 -17157.191} C_VEL
LIN {X 0,Y 284.36,Z 513.689,A -85,B 0,C 180,E1 -17160.378,E2 -17160.378} C_VEL
LIN {X 0,Y 284.38,Z 513.681,A -85,B 0,C 180,E1 -17163.588,E2 -17163.588} C_VEL
LIN {X 0,Y 284.369,Z 513.686,A -85,B 0,C 180,E1 -17166.708,E2 -17166.708} C_VEL
LIN {X 0,Y 284.406,Z 513.678,A -85,B 0,C 180,E1 -17171.263,E2 -17171.263} C_VEL
LIN {X 0,Y 284.495,Z 513.668,A -85,B 0,C 180,E1 -17174.46,E2 -17174.46} C_VEL
LIN {X 0,Y 284.491,Z 513.671,A -85,B 0,C 180,E1 -17178.603,E2 -17178.603} C_VEL
LIN {X 0,Y 284.626,Z 513.654,A -85,B 0,C 180,E1 -17181.481,E2 -17181.481} C_VEL
LIN {X 0,Y 284.599,Z 513.654,A -85,B 0,C 180,E1 -17184.332,E2 -17184.332} C_VEL
LIN {X 0,Y 284.861,Z 513.625,A -85,B 0,C 180,E1 -17188.587,E2 -17188.587} C_VEL
LIN {X 0,Y 284.778,Z 513.636,A -85,B 0,C 180,E1 -17191.415,E2 -17191.415} C_VEL
LIN {X 0,Y 284.236,Z 513.749,A -85,B 0,C 180,E1 -17194.401,E2 -17194.401} C_VEL
LIN {X 0,Y 285.202,Z 516.529,A -85,B 0,C 180,E1 -17194.63,E2 -17194.63} C_VEL
LIN {X 0,Y 287.598,Z 520.869,A -85,B 0,C 180,E1 -17195.096,E2 -17195.096} C_VEL
LIN {X 0,Y 291.417,Z 529.815,A -85,B 0,C 180,E1 -17196.014,E2 -17196.014} C_VEL
LIN {X 0,Y 296.385,Z 543.996,A -85,B 0,C 180,E1 -17197.513,E2 -17197.513} C_VEL
LIN {X 0,Y 299.871,Z 555.972,A -85,B 0,C 180,E1 -17198.882,E2 -17198.882} C_VEL
LIN {X 0,Y 302.14,Z 565.39,A -85,B 0,C 180,E1 -17200.047,E2 -17200.047} C_VEL
LIN {X 0,Y 300.071,Z 578.219,A -85,B 0,C 180,E1 -17201.338,E2 -17201.338} C_VEL
LIN {X 0,Y 297.61,Z 591.387,A -85,B 0,C 180,E1 -17202.965,E2 -17202.965} C_VEL
LIN {X 0,Y 295.129,Z 603.716,A -85,B 0,C 180,E1 -17204.833,E2 -17204.833} C_VEL
LIN {X 0,Y 292.74,Z 614.265,A -85,B 0,C 180,E1 -17206.744,E2 -17206.744} C_VEL
LIN {X 0,Y 290.635,Z 623.41,A -85,B 0,C 180,E1 -17208.731,E2 -17208.731} C_VEL
LIN {X 0,Y 288.561,Z 632.387,A -85,B 0,C 180,E1 -17211.054,E2 -17211.054} C_VEL
LIN {X 0,Y 286.509,Z 641.208,A -85,B 0,C 180,E1 -17213.841,E2 -17213.841} C_VEL
LIN {X 0,Y 285.126,Z 647.583,A -85,B 0,C 180,E1 -17216.339,E2 -17216.339} C_VEL
LIN {X 0,Y 284.09,Z 652.776,A -85,B 0,C 180,E1 -17218.843,E2 -17218.843} C_VEL
LIN {X 0,Y 283.362,Z 656.941,A -85,B 0,C 180,E1 -17221.389,E2 -17221.389} C_VEL
LIN {X 0,Y 282.938,Z 659.184,A -85,B 0,C 180,E1 -17223.125,E2 -17223.125} C_VEL
LIN {X 0,Y 282.588,Z 660.977,A -85,B 0,C 180,E1 -17224.891,E2 -17224.891} C_VEL
LIN {X 0,Y 282.345,Z 662.647,A -85,B 0,C 180,E1 -17227.199,E2 -17227.199} C_VEL
LIN {X 0,Y 282.285,Z 663.73,A -85,B 0,C 180,E1 -17230.34,E2 -17230.34} C_VEL
LIN {X 0,Y 282.36,Z 663.74,A -85,B 0,C 180,E1 -17232.224,E2 -17232.224} C_VEL
LIN {X 0,Y 282.549,Z 663.252,A -85,B 0,C 180,E1 -17234.144,E2 -17234.144} C_VEL
LIN {X 0,Y 282.879,Z 662.185,A -85,B 0,C 180,E1 -17236.095,E2 -17236.095} C_VEL
LIN {X 0,Y 283.665,Z 659.633,A -85,B 0,C 180,E1 -17239.014,E2 -17239.014} C_VEL
LIN {X 0,Y 284.817,Z 655.461,A -85,B 0,C 180,E1 -17242.149,E2 -17242.149} C_VEL
LIN {X 0,Y 286.355,Z 650.371,A -85,B 0,C 180,E1 -17244.96,E2 -17244.96} C_VEL
LIN {X 0,Y 288.259,Z 644.324,A -85,B 0,C 180,E1 -17247.562,E2 -17247.562} C_VEL
LIN {X 0,Y 290.869,Z 635.965,A -85,B 0,C 180,E1 -17250.439,E2 -17250.439} C_VEL
LIN {X 0,Y 293.78,Z 626.75,A -85,B 0,C 180,E1 -17252.965,E2 -17252.965} C_VEL
LIN {X 0,Y 296.893,Z 616.113,A -85,B 0,C 180,E1 -17255.34,E2 -17255.34} C_VEL
LIN {X 0,Y 300.193,Z 604.403,A -85,B 0,C 180,E1 -17257.457,E2 -17257.457} C_VEL
LIN {X 0,Y 303.035,Z 593.192,A -85,B 0,C 180,E1 -17259.148,E2 -17259.148} C_VEL
LIN {X 0,Y 305.974,Z 580.413,A -85,B 0,C 180,E1 -17260.726,E2 -17260.726} C_VEL
LIN {X 0,Y 307.792,Z 571.009,A -85,B 0,C 180,E1 -17261.701,E2 -17261.701} C_VEL
LIN {X 0,Y 305.186,Z 560.016,A -85,B 0,C 180,E1 -17263.382,E2 -17263.382} C_VEL
LIN {X 0,Y 301.841,Z 549.982,A -85,B 0,C 180,E1 -17264.938,E2 -17264.938} C_VEL
LIN {X 0,Y 297.726,Z 540.08,A -85,B 0,C 180,E1 -17266.536,E2 -17266.536} C_VEL
LIN {X 0,Y 292.999,Z 530.583,A -85,B 0,C 180,E1 -17268.148,E2 -17268.148} C_VEL
LIN {X 0,Y 289.881,Z 525.534,A -85,B 0,C 180,E1 -17269.122,E2 -17269.122} C_VEL
LIN {X 0,Y 287.345,Z 522.665,A -85,B 0,C 180,E1 -17269.891,E2 -17269.891} C_VEL
LIN {X 0,Y 282.49,Z 520.026,A -85,B 0,C 180,E1 -17271.105,E2 -17271.105} C_VEL
LIN {X 0,Y 278.116,Z 517.846,A -85,B 0,C 180,E1 -17272.352,E2 -17272.352} C_VEL
LIN {X 0,Y 277.98,Z 516.427,A -85,B 0,C 180,E1 -17277.101,E2 -17277.101} C_VEL
LIN {X 0,Y 278.076,Z 515.722,A -85,B 0,C 180,E1 -17279.999,E2 -17279.999} C_VEL
LIN {X 0,Y 277.808,Z 515.271,A -85,B 0,C 180,E1 -17282.9,E2 -17282.9} C_VEL
LIN {X 0,Y 277.689,Z 514.857,A -85,B 0,C 180,E1 -17287.269,E2 -17287.269} C_VEL
LIN {X 0,Y 277.561,Z 514.833,A -85,B 0,C 180,E1 -17290.209,E2 -17290.209} C_VEL
LIN {X 0,Y 277.523,Z 515.172,A -85,B 0,C 180,E1 -17294.669,E2 -17294.669} C_VEL
LIN {X 0,Y 277.566,Z 515.716,A -85,B 0,C 180,E1 -17297.688,E2 -17297.688} C_VEL
LIN {X 0,Y 277.645,Z 516.5,A -85,B 0,C 180,E1 -17300.755,E2 -17300.755} C_VEL
LIN {X 0,Y 277.891,Z 517.76,A -85,B 0,C 180,E1 -17304.432,E2 -17304.432} C_VEL
LIN {X 0,Y 278.138,Z 519.304,A -85,B 0,C 180,E1 -17307.825,E2 -17307.825} C_VEL
LIN {X 0,Y 278.4,Z 520.98,A -85,B 0,C 180,E1 -17310.874,E2 -17310.874} C_VEL
LIN {X 0,Y 278.922,Z 523.977,A -85,B 0,C 180,E1 -17315.417,E2 -17315.417} C_VEL
LIN {X 0,Y 279.406,Z 526.758,A -85,B 0,C 180,E1 -17318.964,E2 -17318.964} C_VEL
LIN {X 0,Y 279.912,Z 530.079,A -85,B 0,C 180,E1 -17322.68,E2 -17322.68} C_VEL
LIN {X 0,Y 280.266,Z 532.764,A -85,B 0,C 180,E1 -17325.402,E2 -17325.402} C_VEL
LIN {X 0,Y 280.313,Z 534.907,A -85,B 0,C 180,E1 -17327.395,E2 -17327.395} C_VEL
LIN {X 0,Y 280.225,Z 535.941,A -85,B 0,C 180,E1 -17328.175,E2 -17328.175} C_VEL
LIN {X 0,Y 281.216,Z 539.124,A -85,B 0,C 180,E1 -17328.567,E2 -17328.567} C_VEL
LIN {X 0,Y 282.821,Z 542.056,A -85,B 0,C 180,E1 -17329.096,E2 -17329.096} C_VEL
LIN {X 0,Y 284.541,Z 545.988,A -85,B 0,C 180,E1 -17329.691,E2 -17329.691} C_VEL
LIN {X 0,Y 288.652,Z 557.094,A -85,B 0,C 180,E1 -17331.288,E2 -17331.288} C_VEL
LIN {X 0,Y 291.914,Z 567.585,A -85,B 0,C 180,E1 -17332.734,E2 -17332.734} C_VEL
LIN {X 0,Y 294.8,Z 581.099,A -85,B 0,C 180,E1 -17334.494,E2 -17334.494} C_VEL
LIN {X 0,Y 296.407,Z 593.324,A -85,B 0,C 180,E1 -17336.085,E2 -17336.085} C_VEL
LIN {X 0,Y 296.938,Z 606.85,A -85,B 0,C 180,E1 -17337.903,E2 -17337.903} C_VEL
LIN {X 0,Y 296.81,Z 611.855,A -85,B 0,C 180,E1 -17338.605,E2 -17338.605} C_VEL
LIN {X 0,Y 293.619,Z 624.486,A -85,B 0,C 180,E1 -17340.22,E2 -17340.22} C_VEL
LIN {X 0,Y 290.097,Z 637.182,A -85,B 0,C 180,E1 -17342.202,E2 -17342.202} C_VEL
LIN {X 0,Y 286.91,Z 647.893,A -85,B 0,C 180,E1 -17344.227,E2 -17344.227} C_VEL
LIN {X 0,Y 283.777,Z 658.474,A -85,B 0,C 180,E1 -17346.655,E2 -17346.655} C_VEL
LIN {X 0,Y 281.213,Z 667.363,A -85,B 0,C 180,E1 -17349.137,E2 -17349.137} C_VEL
LIN {X 0,Y 279.176,Z 674.845,A -85,B 0,C 180,E1 -17351.658,E2 -17351.658} C_VEL
LIN {X 0,Y 277.33,Z 681.803,A -85,B 0,C 180,E1 -17354.544,E2 -17354.544} C_VEL
LIN {X 0,Y 276.244,Z 687.439,A -85,B 0,C 180,E1 -17357.511,E2 -17357.511} C_VEL
LIN {X 0,Y 275.695,Z 690.719,A -85,B 0,C 180,E1 -17359.72,E2 -17359.72} C_VEL
LIN {X 0,Y 275.374,Z 694.059,A -85,B 0,C 180,E1 -17362.668,E2 -17362.668} C_VEL
LIN {X 0,Y 275.382,Z 696.184,A -85,B 0,C 180,E1 -17365.608,E2 -17365.608} C_VEL
LIN {X 0,Y 275.489,Z 697.08,A -85,B 0,C 180,E1 -17368.537,E2 -17368.537} C_VEL
LIN {X 0,Y 275.62,Z 697.092,A -85,B 0,C 180,E1 -17369.999,E2 -17369.999} C_VEL
LIN {X 0,Y 275.447,Z 696.193,A -85,B 0,C 180,E1 -17372.924,E2 -17372.924} C_VEL
LIN {X 0,Y 275.528,Z 694.096,A -85,B 0,C 180,E1 -17375.855,E2 -17375.855} C_VEL
LIN {X 0,Y 275.555,Z 690.726,A -85,B 0,C 180,E1 -17378.802,E2 -17378.802} C_VEL
LIN {X 0,Y 275.97,Z 686.013,A -85,B 0,C 180,E1 -17381.754,E2 -17381.754} C_VEL
LIN {X 0,Y 276.918,Z 679.843,A -85,B 0,C 180,E1 -17384.701,E2 -17384.701} C_VEL
LIN {X 0,Y 278.47,Z 672.071,A -85,B 0,C 180,E1 -17387.628,E2 -17387.628} C_VEL
LIN {X 0,Y 280.287,Z 663.749,A -85,B 0,C 180,E1 -17390.167,E2 -17390.167} C_VEL
LIN {X 0,Y 282.701,Z 653.769,A -85,B 0,C 180,E1 -17392.663,E2 -17392.663} C_VEL
LIN {X 0,Y 284.956,Z 643.518,A -85,B 0,C 180,E1 -17394.788,E2 -17394.788} C_VEL
LIN {X 0,Y 287.553,Z 632.467,A -85,B 0,C 180,E1 -17396.685,E2 -17396.685} C_VEL
LIN {X 0,Y 290.093,Z 620.565,A -85,B 0,C 180,E1 -17398.387,E2 -17398.387} C_VEL
LIN {X 0,Y 292.375,Z 608.983,A -85,B 0,C 180,E1 -17399.763,E2 -17399.763} C_VEL
LIN {X 0,Y 291.224,Z 595.886,A -85,B 0,C 180,E1 -17401.362,E2 -17401.362} C_VEL
LIN {X 0,Y 289.256,Z 582.389,A -85,B 0,C 180,E1 -17402.834,E2 -17402.834} C_VEL
LIN {X 0,Y 286.164,Z 567.063,A -85,B 0,C 180,E1 -17404.318,E2 -17404.318} C_VEL
LIN {X 0,Y 282.456,Z 552.993,A -85,B 0,C 180,E1 -17405.534,E2 -17405.534} C_VEL
LIN {X 0,Y 278.875,Z 541.241,A -85,B 0,C 180,E1 -17406.446,E2 -17406.446} C_VEL
LIN {X 0,Y 278.824,Z 540.709,A -85,B 0,C 180,E1 -17406.496,E2 -17406.496} C_VEL
LIN {X 0,Y 279.813,Z 535.002,A -85,B 0,C 180,E1 -17410.769,E2 -17410.769} C_VEL
LIN {X 0,Y 280.203,Z 531.716,A -85,B 0,C 180,E1 -17413.334,E2 -17413.334} C_VEL
LIN {X 0,Y 279.918,Z 529.301,A -85,B 0,C 180,E1 -17415.332,E2 -17415.332} C_VEL
LIN {X 0,Y 279.063,Z 525.019,A -85,B 0,C 180,E1 -17419.097,E2 -17419.097} C_VEL
LIN {X 0,Y 278.343,Z 521.154,A -85,B 0,C 180,E1 -17422.701,E2 -17422.701} C_VEL
LIN {X 0,Y 277.702,Z 517.2,A -85,B 0,C 180,E1 -17426.629,E2 -17426.629} C_VEL
LIN {X 0,Y 277.279,Z 514.57,A -85,B 0,C 180,E1 -17429.541,E2 -17429.541} C_VEL
LIN {X 0,Y 277.352,Z 514.561,A -85,B 0,C 180,E1 -17432.864,E2 -17432.864} C_VEL
LIN {X 0,Y 277.289,Z 514.57,A -85,B 0,C 180,E1 -17436.076,E2 -17436.076} C_VEL
LIN {X 0,Y 277.337,Z 514.563,A -85,B 0,C 180,E1 -17440.766,E2 -17440.766} C_VEL
LIN {X 0,Y 277.427,Z 514.553,A -85,B 0,C 180,E1 -17445.326,E2 -17445.326} C_VEL
LIN {X 0,Y 277.499,Z 514.532,A -85,B 0,C 180,E1 -17449.789,E2 -17449.789} C_VEL
LIN {X 0,Y 277.645,Z 514.517,A -85,B 0,C 180,E1 -17452.729,E2 -17452.729} C_VEL
LIN {X 0,Y 277.817,Z 514.497,A -85,B 0,C 180,E1 -17458.551,E2 -17458.551} C_VEL
LIN {X 0,Y 277.815,Z 514.489,A -85,B 0,C 180,E1 -17461.45,E2 -17461.45} C_VEL
LIN {X 0,Y 277.635,Z 514.527,A -85,B 0,C 180,E1 -17467.272,E2 -17467.272} C_VEL
LIN {X 0,Y 277.453,Z 514.538,A -85,B 0,C 180,E1 -17470.214,E2 -17470.214} C_VEL
LIN {X 0,Y 277.421,Z 514.544,A -85,B 0,C 180,E1 -17474.676,E2 -17474.676} C_VEL
LIN {X 0,Y 277.338,Z 514.563,A -85,B 0,C 180,E1 -17479.235,E2 -17479.235} C_VEL
LIN {X 0,Y 277.313,Z 514.548,A -85,B 0,C 180,E1 -17484.171,E2 -17484.171} C_VEL
LIN {X 0,Y 277.321,Z 514.562,A -85,B 0,C 180,E1 -17487.507,E2 -17487.507} C_VEL
LIN {X 0,Y 277.267,Z 514.57,A -85,B 0,C 180,E1 -17490.483,E2 -17490.483} C_VEL
LIN {X 0,Y 277.25,Z 514.562,A -85,B 0,C 180,E1 -17493.896,E2 -17493.896} C_VEL
LIN {X 0,Y 277.287,Z 514.56,A -85,B 0,C 180,E1 -17497.467,E2 -17497.467} C_VEL
LIN {X 0,Y 277.292,Z 514.569,A -85,B 0,C 180,E1 -17501.223,E2 -17501.223} C_VEL
LIN {X 0,Y 277.286,Z 514.561,A -85,B 0,C 180,E1 -17505.21,E2 -17505.21} C_VEL
LIN {X 0,Y 277.294,Z 514.569,A -85,B 0,C 180,E1 -17509.496,E2 -17509.496} C_VEL
LIN {X 0,Y 277.29,Z 514.568,A -85,B 0,C 180,E1 -17512.536,E2 -17512.536} C_VEL
LIN {X 0,Y 277.254,Z 514.567,A -85,B 0,C 180,E1 -17516.107,E2 -17516.107} C_VEL
LIN {X 0,Y 277.262,Z 514.577,A -85,B 0,C 180,E1 -17519.54,E2 -17519.54} C_VEL
LIN {X 0,Y 277.36,Z 514.555,A -85,B 0,C 180,E1 -17522.866,E2 -17522.866} C_VEL
LIN {X 0,Y 277.34,Z 514.564,A -85,B 0,C 180,E1 -17526.082,E2 -17526.082} C_VEL
LIN {X 0,Y 277.348,Z 514.555,A -85,B 0,C 180,E1 -17530.768,E2 -17530.768} C_VEL
LIN {X 0,Y 277.438,Z 514.547,A -85,B 0,C 180,E1 -17535.327,E2 -17535.327} C_VEL
LIN {X 0,Y 277.464,Z 514.544,A -85,B 0,C 180,E1 -17539.788,E2 -17539.788} C_VEL
LIN {X 0,Y 277.633,Z 514.526,A -85,B 0,C 180,E1 -17542.729,E2 -17542.729} C_VEL
LIN {X 0,Y 277.827,Z 514.502,A -85,B 0,C 180,E1 -17548.551,E2 -17548.551} C_VEL
LIN {X 0,Y 277.734,Z 514.513,A -85,B 0,C 180,E1 -17551.451,E2 -17551.451} C_VEL
LIN {X 0,Y 277.261,Z 514.572,A -85,B 0,C 180,E1 -17553.543,E2 -17553.543} C_VEL
LIN {X 0,Y 278.281,Z 517.505,A -85,B 0,C 180,E1 -17553.802,E2 -17553.802} C_VEL
LIN {X 0,Y 283.56,Z 527.762,A -85,B 0,C 180,E1 -17554.955,E2 -17554.955} C_VEL
LIN {X 0,Y 288.502,Z 541.223,A -85,B 0,C 180,E1 -17556.415,E2 -17556.415} C_VEL
LIN {X 0,Y 292.589,Z 554.559,A -85,B 0,C 180,E1 -17557.984,E2 -17557.984} C_VEL
LIN {X 0,Y 295.618,Z 567.13,A -85,B 0,C 180,E1 -17559.58,E2 -17559.58} C_VEL
LIN {X 0,Y 293.222,Z 581.07,A -85,B 0,C 180,E1 -17561.055,E2 -17561.055} C_VEL
LIN {X 0,Y 290.668,Z 593.916,A -85,B 0,C 180,E1 -17562.729,E2 -17562.729} C_VEL
LIN {X 0,Y 288.102,Z 606.028,A -85,B 0,C 180,E1 -17564.661,E2 -17564.661} C_VEL
LIN {X 0,Y 285.443,Z 617.07,A -85,B 0,C 180,E1 -17566.78,E2 -17566.78} C_VEL
LIN {X 0,Y 282.919,Z 627.677,A -85,B 0,C 180,E1 -17569.27,E2 -17569.27} C_VEL
LIN {X 0,Y 280.914,Z 636.044,A -85,B 0,C 180,E1 -17571.656,E2 -17571.656} C_VEL
LIN {X 0,Y 279.139,Z 643.636,A -85,B 0,C 180,E1 -17574.283,E2 -17574.283} C_VEL
LIN {X 0,Y 277.684,Z 650.201,A -85,B 0,C 180,E1 -17577.102,E2 -17577.102} C_VEL
LIN {X 0,Y 276.598,Z 655.84,A -85,B 0,C 180,E1 -17580.242,E2 -17580.242} C_VEL
LIN {X 0,Y 275.934,Z 659.325,A -85,B 0,C 180,E1 -17582.805,E2 -17582.805} C_VEL
LIN {X 0,Y 275.364,Z 662.281,A -85,B 0,C 180,E1 -17585.946,E2 -17585.946} C_VEL
LIN {X 0,Y 275.22,Z 663.405,A -85,B 0,C 180,E1 -17587.797,E2 -17587.797} C_VEL
LIN {X 0,Y 275.193,Z 664.094,A -85,B 0,C 180,E1 -17589.989,E2 -17589.989} C_VEL
LIN {X 0,Y 275.286,Z 664.187,A -85,B 0,C 180,E1 -17592.236,E2 -17592.236} C_VEL
LIN {X 0,Y 275.677,Z 663.113,A -85,B 0,C 180,E1 -17595.547,E2 -17595.547} C_VEL
LIN {X 0,Y 276.481,Z 660.781,A -85,B 0,C 180,E1 -17598.63,E2 -17598.63} C_VEL
LIN {X 0,Y 277.554,Z 657.13,A -85,B 0,C 180,E1 -17601.717,E2 -17601.717} C_VEL
LIN {X 0,Y 279.038,Z 652.428,A -85,B 0,C 180,E1 -17604.598,E2 -17604.598} C_VEL
LIN {X 0,Y 281.004,Z 646.573,A -85,B 0,C 180,E1 -17607.368,E2 -17607.368} C_VEL
LIN {X 0,Y 283.504,Z 639.045,A -85,B 0,C 180,E1 -17610.185,E2 -17610.185} C_VEL
LIN {X 0,Y 286.265,Z 630.698,A -85,B 0,C 180,E1 -17612.7,E2 -17612.7} C_VEL
LIN {X 0,Y 289.331,Z 621.233,A -85,B 0,C 180,E1 -17615.037,E2 -17615.037} C_VEL
LIN {X 0,Y 292.485,Z 610.741,A -85,B 0,C 180,E1 -17617.179,E2 -17617.179} C_VEL
LIN {X 0,Y 295.75,Z 599.154,A -85,B 0,C 180,E1 -17619.117,E2 -17619.117} C_VEL
LIN {X 0,Y 298.801,Z 587.139,A -85,B 0,C 180,E1 -17620.774,E2 -17620.774} C_VEL
LIN {X 0,Y 301.788,Z 572.936,A -85,B 0,C 180,E1 -17622.377,E2 -17622.377} C_VEL
LIN {X 0,Y 299.202,Z 561.755,A -85,B 0,C 180,E1 -17624.183,E2 -17624.183} C_VEL
LIN {X 0,Y 295.02,Z 549.451,A -85,B 0,C 180,E1 -17626.218,E2 -17626.218} C_VEL
LIN {X 0,Y 290.101,Z 538.39,A -85,B 0,C 180,E1 -17628.168,E2 -17628.168} C_VEL
LIN {X 0,Y 286.005,Z 530.922,A -85,B 0,C 180,E1 -17629.621,E2 -17629.621} C_VEL
LIN {X 0,Y 283.413,Z 526.658,A -85,B 0,C 180,E1 -17630.503,E2 -17630.503} C_VEL
LIN {X 0,Y 281.411,Z 523.221,A -85,B 0,C 180,E1 -17631.189,E2 -17631.189} C_VEL
LIN {X 0,Y 278.839,Z 519.922,A -85,B 0,C 180,E1 -17632.031,E2 -17632.031} C_VEL
LIN {X 0,Y 278.116,Z 517.846,A -85,B 0,C 180,E1 -17632.352,E2 -17632.352} C_VEL
LIN {X 0,Y 277.574,Z 517.661,A -85,B 0,C 180,E1 -17633.129,E2 -17633.129} C_VEL
LIN {X 0,Y 275.538,Z 517.586,A -85,B 0,C 180,E1 -17634.703,E2 -17634.703} C_VEL
LIN {X 0,Y 272.111,Z 517.742,A -85,B 0,C 180,E1 -17637.108,E2 -17637.108} C_VEL
LIN {X 0,Y 271.103,Z 517.448,A -85,B 0,C 180,E1 -17638.78,E2 -17638.78} C_VEL
LIN {X 0,Y 271.023,Z 516.949,A -85,B 0,C 180,E1 -17641.485,E2 -17641.485} C_VEL
LIN {X 0,Y 270.75,Z 516.402,A -85,B 0,C 180,E1 -17647.457,E2 -17647.457} C_VEL
LIN {X 0,Y 270.62,Z 516.42,A -85,B 0,C 180,E1 -17650.473,E2 -17650.473} C_VEL
LIN {X 0,Y 270.63,Z 516.833,A -85,B 0,C 180,E1 -17655.051,E2 -17655.051} C_VEL
LIN {X 0,Y 270.71,Z 517.813,A -85,B 0,C 180,E1 -17659.724,E2 -17659.724} C_VEL
LIN {X 0,Y 270.991,Z 519.523,A -85,B 0,C 180,E1 -17664.81,E2 -17664.81} C_VEL
LIN {X 0,Y 271.248,Z 521.102,A -85,B 0,C 180,E1 -17668.245,E2 -17668.245} C_VEL
LIN {X 0,Y 271.494,Z 522.815,A -85,B 0,C 180,E1 -17671.323,E2 -17671.323} C_VEL
LIN {X 0,Y 271.866,Z 524.971,A -85,B 0,C 180,E1 -17674.661,E2 -17674.661} C_VEL
LIN {X 0,Y 272.354,Z 527.638,A -85,B 0,C 180,E1 -17678.265,E2 -17678.265} C_VEL
LIN {X 0,Y 272.827,Z 530.857,A -85,B 0,C 180,E1 -17682.048,E2 -17682.048} C_VEL
LIN {X 0,Y 273.316,Z 534.692,A -85,B 0,C 180,E1 -17686.031,E2 -17686.031} C_VEL
LIN {X 0,Y 273.376,Z 535.109,A -85,B 0,C 180,E1 -17686.372,E2 -17686.372} C_VEL
LIN {X 0,Y 274.511,Z 538.482,A -85,B 0,C 180,E1 -17686.857,E2 -17686.857} C_VEL
LIN {X 0,Y 276.294,Z 541.373,A -85,B 0,C 180,E1 -17687.489,E2 -17687.489} C_VEL
LIN {X 0,Y 278.049,Z 545.448,A -85,B 0,C 180,E1 -17688.165,E2 -17688.165} C_VEL
LIN {X 0,Y 282.079,Z 555.524,A -85,B 0,C 180,E1 -17689.795,E2 -17689.795} C_VEL
LIN {X 0,Y 285.909,Z 567.997,A -85,B 0,C 180,E1 -17691.635,E2 -17691.635} C_VEL
LIN {X 0,Y 288.514,Z 579.753,A -85,B 0,C 180,E1 -17693.277,E2 -17693.277} C_VEL
LIN {X 0,Y 290.368,Z 593.696,A -85,B 0,C 180,E1 -17695.194,E2 -17695.194} C_VEL
LIN {X 0,Y 290.869,Z 607.022,A -85,B 0,C 180,E1 -17697.068,E2 -17697.068} C_VEL
LIN {X 0,Y 290.508,Z 613.798,A -85,B 0,C 180,E1 -17698.047,E2 -17698.047} C_VEL
LIN {X 0,Y 286.845,Z 627.173,A -85,B 0,C 180,E1 -17699.849,E2 -17699.849} C_VEL
LIN {X 0,Y 283.211,Z 639.361,A -85,B 0,C 180,E1 -17701.869,E2 -17701.869} C_VEL
LIN {X 0,Y 279.5,Z 651.229,A -85,B 0,C 180,E1 -17704.294,E2 -17704.294} C_VEL
LIN {X 0,Y 276.455,Z 661.168,A -85,B 0,C 180,E1 -17706.794,E2 -17706.794} C_VEL
LIN {X 0,Y 273.482,Z 670.61,A -85,B 0,C 180,E1 -17709.7,E2 -17709.7} C_VEL
LIN {X 0,Y 271.314,Z 678.339,A -85,B 0,C 180,E1 -17712.669,E2 -17712.669} C_VEL
LIN {X 0,Y 269.749,Z 684.562,A -85,B 0,C 180,E1 -17715.669,E2 -17715.669} C_VEL
LIN {X 0,Y 268.776,Z 689.417,A -85,B 0,C 180,E1 -17718.69,E2 -17718.69} C_VEL
LIN {X 0,Y 268.416,Z 692.198,A -85,B 0,C 180,E1 -17720.961,E2 -17720.961} C_VEL
LIN {X 0,Y 268.34,Z 695.152,A -85,B 0,C 180,E1 -17724.406,E2 -17724.406} C_VEL
LIN {X 0,Y 268.357,Z 696.379,A -85,B 0,C 180,E1 -17726.997,E2 -17726.997} C_VEL
LIN {X 0,Y 268.531,Z 696.648,A -85,B 0,C 180,E1 -17729.999,E2 -17729.999} C_VEL
LIN {X 0,Y 268.375,Z 695.709,A -85,B 0,C 180,E1 -17733.001,E2 -17733.001} C_VEL
LIN {X 0,Y 268.426,Z 693.567,A -85,B 0,C 180,E1 -17736.011,E2 -17736.011} C_VEL
LIN {X 0,Y 268.47,Z 690.148,A -85,B 0,C 180,E1 -17739.036,E2 -17739.036} C_VEL
LIN {X 0,Y 268.963,Z 685.392,A -85,B 0,C 180,E1 -17742.065,E2 -17742.065} C_VEL
LIN {X 0,Y 269.967,Z 679.168,A -85,B 0,C 180,E1 -17745.088,E2 -17745.088} C_VEL
LIN {X 0,Y 271.592,Z 671.317,A -85,B 0,C 180,E1 -17748.09,E2 -17748.09} C_VEL
LIN {X 0,Y 273.569,Z 662.951,A -85,B 0,C 180,E1 -17750.684,E2 -17750.684} C_VEL
LIN {X 0,Y 275.959,Z 653.291,A -85,B 0,C 180,E1 -17753.144,E2 -17753.144} C_VEL
LIN {X 0,Y 278.433,Z 642.552,A -85,B 0,C 180,E1 -17755.409,E2 -17755.409} C_VEL
LIN {X 0,Y 281.361,Z 630.314,A -85,B 0,C 180,E1 -17757.522,E2 -17757.522} C_VEL
LIN {X 0,Y 284.096,Z 618.079,A -85,B 0,C 180,E1 -17759.246,E2 -17759.246} C_VEL
LIN {X 0,Y 285.632,Z 610.65,A -85,B 0,C 180,E1 -17760.144,E2 -17760.144} C_VEL
LIN {X 0,Y 284.877,Z 599.392,A -85,B 0,C 180,E1 -17761.579,E2 -17761.579} C_VEL
LIN {X 0,Y 283.04,Z 585.392,A -85,B 0,C 180,E1 -17763.204,E2 -17763.204} C_VEL
LIN {X 0,Y 280.327,Z 571.039,A -85,B 0,C 180,E1 -17764.691,E2 -17764.691} C_VEL
LIN {X 0,Y 276.81,Z 556.663,A -85,B 0,C 180,E1 -17766.019,E2 -17766.019} C_VEL
LIN {X 0,Y 272.012,Z 540.942,A -85,B 0,C 180,E1 -17767.332,E2 -17767.332} C_VEL
LIN {X 0,Y 271.965,Z 540.294,A -85,B 0,C 180,E1 -17767.408,E2 -17767.408} C_VEL
LIN {X 0,Y 272.597,Z 536.716,A -85,B 0,C 180,E1 -17770.129,E2 -17770.129} C_VEL
LIN {X 0,Y 273.13,Z 533.207,A -85,B 0,C 180,E1 -17772.937,E2 -17772.937} C_VEL
LIN {X 0,Y 272.975,Z 530.749,A -85,B 0,C 180,E1 -17774.981,E2 -17774.981} C_VEL
LIN {X 0,Y 272.212,Z 526.827,A -85,B 0,C 180,E1 -17778.478,E2 -17778.478} C_VEL
LIN {X 0,Y 271.576,Z 523.51,A -85,B 0,C 180,E1 -17781.605,E2 -17781.605} C_VEL
LIN {X 0,Y 270.828,Z 518.991,A -85,B 0,C 180,E1 -17786.137,E2 -17786.137} C_VEL
LIN {X 0,Y 270.237,Z 515.446,A -85,B 0,C 180,E1 -17790.055,E2 -17790.055} C_VEL
LIN {X 0,Y 270.254,Z 515.447,A -85,B 0,C 180,E1 -17793.763,E2 -17793.763} C_VEL
LIN {X 0,Y 270.202,Z 515.454,A -85,B 0,C 180,E1 -17797.037,E2 -17797.037} C_VEL
LIN {X 0,Y 270.293,Z 515.441,A -85,B 0,C 180,E1 -17800.244,E2 -17800.244} C_VEL
LIN {X 0,Y 270.395,Z 515.427,A -85,B 0,C 180,E1 -17804.935,E2 -17804.935} C_VEL
LIN {X 0,Y 270.434,Z 515.413,A -85,B 0,C 180,E1 -17809.519,E2 -17809.519} C_VEL
LIN {X 0,Y 270.603,Z 515.393,A -85,B 0,C 180,E1 -17812.539,E2 -17812.539} C_VEL
LIN {X 0,Y 270.783,Z 515.372,A -85,B 0,C 180,E1 -17818.513,E2 -17818.513} C_VEL
LIN {X 0,Y 270.781,Z 515.364,A -85,B 0,C 180,E1 -17821.488,E2 -17821.488} C_VEL
LIN {X 0,Y 270.592,Z 515.405,A -85,B 0,C 180,E1 -17827.462,E2 -17827.462} C_VEL
LIN {X 0,Y 270.405,Z 515.414,A -85,B 0,C 180,E1 -17830.483,E2 -17830.483} C_VEL
LIN {X 0,Y 270.389,Z 515.42,A -85,B 0,C 180,E1 -17835.066,E2 -17835.066} C_VEL
LIN {X 0,Y 270.295,Z 515.438,A -85,B 0,C 180,E1 -17839.757,E2 -17839.757} C_VEL
LIN {X 0,Y 270.268,Z 515.424,A -85,B 0,C 180,E1 -17844.587,E2 -17844.587} C_VEL
LIN {X 0,Y 270.265,Z 515.443,A -85,B 0,C 180,E1 -17847.91,E2 -17847.91} C_VEL
LIN {X 0,Y 270.18,Z 515.456,A -85,B 0,C 180,E1 -17851.349,E2 -17851.349} C_VEL
LIN {X 0,Y 270.212,Z 515.436,A -85,B 0,C 180,E1 -17854.905,E2 -17854.905} C_VEL
LIN {X 0,Y 270.219,Z 515.444,A -85,B 0,C 180,E1 -17858.719,E2 -17858.719} C_VEL
LIN {X 0,Y 270.254,Z 515.443,A -85,B 0,C 180,E1 -17862.543,E2 -17862.543} C_VEL
LIN {X 0,Y 270.231,Z 515.434,A -85,B 0,C 180,E1 -17866.737,E2 -17866.737} C_VEL
LIN {X 0,Y 270.246,Z 515.446,A -85,B 0,C 180,E1 -17869.449,E2 -17869.449} C_VEL
LIN {X 0,Y 270.257,Z 515.441,A -85,B 0,C 180,E1 -17873.723,E2 -17873.723} C_VEL
LIN {X 0,Y 270.204,Z 515.445,A -85,B 0,C 180,E1 -17876.894,E2 -17876.894} C_VEL
LIN {X 0,Y 270.23,Z 515.45,A -85,B 0,C 180,E1 -17880.388,E2 -17880.388} C_VEL
LIN {X 0,Y 270.268,Z 515.437,A -85,B 0,C 180,E1 -17883.766,E2 -17883.766} C_VEL
LIN {X 0,Y 270.239,Z 515.448,A -85,B 0,C 180,E1 -17887.041,E2 -17887.041} C_VEL
LIN {X 0,Y 270.304,Z 515.432,A -85,B 0,C 180,E1 -17890.246,E2 -17890.246} C_VEL
LIN {X 0,Y 270.406,Z 515.423,A -85,B 0,C 180,E1 -17894.937,E2 -17894.937} C_VEL
LIN {X 0,Y 270.416,Z 515.424,A -85,B 0,C 180,E1 -17899.519,E2 -17899.519} C_VEL
LIN {X 0,Y 270.59,Z 515.403,A -85,B 0,C 180,E1 -17902.539,E2 -17902.539} C_VEL
LIN {X 0,Y 270.793,Z 515.378,A -85,B 0,C 180,E1 -17908.514,E2 -17908.514} C_VEL
LIN {X 0,Y 270.69,Z 515.391,A -85,B 0,C 180,E1 -17911.488,E2 -17911.488} C_VEL
LIN {X 0,Y 270.379,Z 515.431,A -85,B 0,C 180,E1 -17912.654,E2 -17912.654} C_VEL
LIN {X 0,Y 271.276,Z 518.203,A -85,B 0,C 180,E1 -17912.901,E2 -17912.901} C_VEL
LIN {X 0,Y 277.897,Z 531.316,A -85,B 0,C 180,E1 -17914.467,E2 -17914.467} C_VEL
LIN {X 0,Y 282.671,Z 544.725,A -85,B 0,C 180,E1 -17915.998,E2 -17915.998} C_VEL
LIN {X 0,Y 286.708,Z 558.335,A -85,B 0,C 180,E1 -17917.687,E2 -17917.687} C_VEL
LIN {X 0,Y 289.079,Z 568.768,A -85,B 0,C 180,E1 -17919.08,E2 -17919.08} C_VEL
LIN {X 0,Y 286.645,Z 582.343,A -85,B 0,C 180,E1 -17920.568,E2 -17920.568} C_VEL
LIN {X 0,Y 283.931,Z 595.391,A -85,B 0,C 180,E1 -17922.327,E2 -17922.327} C_VEL
LIN {X 0,Y 281.36,Z 607.014,A -85,B 0,C 180,E1 -17924.245,E2 -17924.245} C_VEL
LIN {X 0,Y 278.538,Z 618.366,A -85,B 0,C 180,E1 -17926.5,E2 -17926.5} C_VEL
LIN {X 0,Y 276.071,Z 628.414,A -85,B 0,C 180,E1 -17928.941,E2 -17928.941} C_VEL
LIN {X 0,Y 273.792,Z 637.492,A -85,B 0,C 180,E1 -17931.631,E2 -17931.631} C_VEL
LIN {X 0,Y 271.95,Z 645.137,A -85,B 0,C 180,E1 -17934.424,E2 -17934.424} C_VEL
LIN {X 0,Y 270.641,Z 650.871,A -85,B 0,C 180,E1 -17937.003,E2 -17937.003} C_VEL
LIN {X 0,Y 269.666,Z 655.661,A -85,B 0,C 180,E1 -17939.682,E2 -17939.682} C_VEL
LIN {X 0,Y 268.95,Z 659.276,A -85,B 0,C 180,E1 -17942.335,E2 -17942.335} C_VEL
LIN {X 0,Y 268.303,Z 662.522,A -85,B 0,C 180,E1 -17945.705,E2 -17945.705} C_VEL
LIN {X 0,Y 268.089,Z 664.257,A -85,B 0,C 180,E1 -17948.989,E2 -17948.989} C_VEL
LIN {X 0,Y 268.136,Z 664.66,A -85,B 0,C 180,E1 -17950.94,E2 -17950.94} C_VEL
LIN {X 0,Y 268.273,Z 664.578,A -85,B 0,C 180,E1 -17952.932,E2 -17952.932} C_VEL
LIN {X 0,Y 268.497,Z 663.921,A -85,B 0,C 180,E1 -17955.029,E2 -17955.029} C_VEL
LIN {X 0,Y 268.988,Z 662.673,A -85,B 0,C 180,E1 -17957.209,E2 -17957.209} C_VEL
LIN {X 0,Y 269.957,Z 659.793,A -85,B 0,C 180,E1 -17960.362,E2 -17960.362} C_VEL
LIN {X 0,Y 271.318,Z 655.687,A -85,B 0,C 180,E1 -17963.431,E2 -17963.431} C_VEL
LIN {X 0,Y 273.221,Z 650.163,A -85,B 0,C 180,E1 -17966.495,E2 -17966.495} C_VEL
LIN {X 0,Y 275.577,Z 643.569,A -85,B 0,C 180,E1 -17969.332,E2 -17969.332} C_VEL
LIN {X 0,Y 278.386,Z 635.6,A -85,B 0,C 180,E1 -17972.078,E2 -17972.078} C_VEL
LIN {X 0,Y 281.468,Z 626.702,A -85,B 0,C 180,E1 -17974.565,E2 -17974.565} C_VEL
LIN {X 0,Y 284.891,Z 616.265,A -85,B 0,C 180,E1 -17976.944,E2 -17976.944} C_VEL
LIN {X 0,Y 288.122,Z 605.772,A -85,B 0,C 180,E1 -17978.912,E2 -17978.912} C_VEL
LIN {X 0,Y 291.607,Z 593.339,A -85,B 0,C 180,E1 -17980.829,E2 -17980.829} C_VEL
LIN {X 0,Y 294.821,Z 580.362,A -85,B 0,C 180,E1 -17982.463,E2 -17982.463} C_VEL
LIN {X 0,Y 295.915,Z 575.551,A -85,B 0,C 180,E1 -17982.986,E2 -17982.986} C_VEL
LIN {X 0,Y 293.672,Z 565.18,A -85,B 0,C 180,E1 -17984.737,E2 -17984.737} C_VEL
LIN {X 0,Y 290.056,Z 553.682,A -85,B 0,C 180,E1 -17986.756,E2 -17986.756} C_VEL
LIN {X 0,Y 285.768,Z 543.446,A -85,B 0,C 180,E1 -17988.653,E2 -17988.653} C_VEL
LIN {X 0,Y 281.472,Z 535.334,A -85,B 0,C 180,E1 -17990.33,E2 -17990.33} C_VEL
LIN {X 0,Y 279.467,Z 531.872,A -85,B 0,C 180,E1 -17991.088,E2 -17991.088} C_VEL
LIN {X 0,Y 277.183,Z 528.015,A -85,B 0,C 180,E1 -17991.954,E2 -17991.954} C_VEL
LIN {X 0,Y 274.989,Z 524.805,A -85,B 0,C 180,E1 -17992.75,E2 -17992.75} C_VEL
LIN {X 0,Y 274.3,Z 523.617,A -85,B 0,C 180,E1 -17993.009,E2 -17993.009} C_VEL
LIN {X 0,Y 272.077,Z 521.244,A -85,B 0,C 180,E1 -17993.79,E2 -17993.79} C_VEL
LIN {X 0,Y 271.035,Z 518.595,A -85,B 0,C 180,E1 -17994.326,E2 -17994.326} C_VEL
LIN {X 0,Y 271.103,Z 517.448,A -85,B 0,C 180,E1 -17998.78,E2 -17998.78} C_VEL
LIN {X 0,Y 270.761,Z 517.351,A -85,B 0,C 180,E1 -17999.61,E2 -17999.61} C_VEL
LIN {X 0,Y 269.34,Z 517.427,A -85,B 0,C 180,E1 -18000.832,E2 -18000.832} C_VEL
LIN {X 0,Y 264.846,Z 517.99,A -85,B 0,C 180,E1 -18003.676,E2 -18003.676} C_VEL
LIN {X 0,Y 263.8,Z 518.098,A -85,B 0,C 180,E1 -18004.952,E2 -18004.952} C_VEL
LIN {X 0,Y 263.734,Z 518.081,A -85,B 0,C 180,E1 -18005.385,E2 -18005.385} C_VEL
LIN {X 0,Y 263.82,Z 517.954,A -85,B 0,C 180,E1 -18009.197,E2 -18009.197} C_VEL
LIN {X 0,Y 263.672,Z 518.291,A -85,B 0,C 180,E1 -18013.879,E2 -18013.879} C_VEL
LIN {X 0,Y 263.736,Z 518.804,A -85,B 0,C 180,E1 -18017.045,E2 -18017.045} C_VEL
LIN {X 0,Y 263.836,Z 519.865,A -85,B 0,C 180,E1 -18021.201,E2 -18021.201} C_VEL
LIN {X 0,Y 264.103,Z 521.301,A -85,B 0,C 180,E1 -18025.209,E2 -18025.209} C_VEL
LIN {X 0,Y 264.35,Z 522.92,A -85,B 0,C 180,E1 -18028.678,E2 -18028.678} C_VEL
LIN {X 0,Y 264.623,Z 524.831,A -85,B 0,C 180,E1 -18032.084,E2 -18032.084} C_VEL
LIN {X 0,Y 265.038,Z 527.18,A -85,B 0,C 180,E1 -18035.688,E2 -18035.688} C_VEL
LIN {X 0,Y 265.599,Z 530.371,A -85,B 0,C 180,E1 -18039.882,E2 -18039.882} C_VEL
LIN {X 0,Y 266.131,Z 534.251,A -85,B 0,C 180,E1 -18044.212,E2 -18044.212} C_VEL
LIN {X 0,Y 267.268,Z 537.491,A -85,B 0,C 180,E1 -18044.757,E2 -18044.757} C_VEL
LIN {X 0,Y 269.763,Z 540.923,A -85,B 0,C 180,E1 -18045.717,E2 -18045.717} C_VEL
LIN {X 0,Y 271.515,Z 544.848,A -85,B 0,C 180,E1 -18046.448,E2 -18046.448} C_VEL
LIN {X 0,Y 272.573,Z 546.992,A -85,B 0,C 180,E1 -18046.886,E2 -18046.886} C_VEL
LIN {X 0,Y 274.707,Z 552.305,A -85,B 0,C 180,E1 -18047.827,E2 -18047.827} C_VEL
LIN {X 0,Y 277.763,Z 560.866,A -85,B 0,C 180,E1 -18049.267,E2 -18049.267} C_VEL
LIN {X 0,Y 280.722,Z 571.283,A -85,B 0,C 180,E1 -18050.904,E2 -18050.904} C_VEL
LIN {X 0,Y 283.292,Z 584.412,A -85,B 0,C 180,E1 -18052.841,E2 -18052.841} C_VEL
LIN {X 0,Y 284.597,Z 597.261,A -85,B 0,C 180,E1 -18054.723,E2 -18054.723} C_VEL
LIN {X 0,Y 284.706,Z 610.468,A -85,B 0,C 180,E1 -18056.685,E2 -18056.685} C_VEL
LIN {X 0,Y 284.443,Z 614.725,A -85,B 0,C 180,E1 -18057.329,E2 -18057.329} C_VEL
LIN {X 0,Y 280.744,Z 627.56,A -85,B 0,C 180,E1 -18059.123,E2 -18059.123} C_VEL
LIN {X 0,Y 276.961,Z 639.56,A -85,B 0,C 180,E1 -18061.175,E2 -18061.175} C_VEL
LIN {X 0,Y 273.603,Z 649.781,A -85,B 0,C 180,E1 -18063.287,E2 -18063.287} C_VEL
LIN {X 0,Y 270.264,Z 659.869,A -85,B 0,C 180,E1 -18065.822,E2 -18065.822} C_VEL
LIN {X 0,Y 267.489,Z 668.334,A -85,B 0,C 180,E1 -18068.417,E2 -18068.417} C_VEL
LIN {X 0,Y 265.019,Z 676.377,A -85,B 0,C 180,E1 -18071.444,E2 -18071.444} C_VEL
LIN {X 0,Y 263.131,Z 682.888,A -85,B 0,C 180,E1 -18074.508,E2 -18074.508} C_VEL
LIN {X 0,Y 261.984,Z 688.014,A -85,B 0,C 180,E1 -18077.607,E2 -18077.607} C_VEL
LIN {X 0,Y 261.367,Z 691.867,A -85,B 0,C 180,E1 -18080.715,E2 -18080.715} C_VEL
LIN {X 0,Y 261.213,Z 694.514,A -85,B 0,C 180,E1 -18083.821,E2 -18083.821} C_VEL
LIN {X 0,Y 261.283,Z 695.977,A -85,B 0,C 180,E1 -18086.915,E2 -18086.915} C_VEL
LIN {X 0,Y 261.441,Z 696.206,A -85,B 0,C 180,E1 -18089.999,E2 -18089.999} C_VEL
LIN {X 0,Y 261.304,Z 695.223,A -85,B 0,C 180,E1 -18093.083,E2 -18093.083} C_VEL
LIN {X 0,Y 261.343,Z 693.031,A -85,B 0,C 180,E1 -18096.174,E2 -18096.174} C_VEL
LIN {X 0,Y 261.409,Z 689.561,A -85,B 0,C 180,E1 -18099.282,E2 -18099.282} C_VEL
LIN {X 0,Y 261.961,Z 684.751,A -85,B 0,C 180,E1 -18102.393,E2 -18102.393} C_VEL
LIN {X 0,Y 263.029,Z 678.468,A -85,B 0,C 180,E1 -18105.496,E2 -18105.496} C_VEL
LIN {X 0,Y 264.746,Z 670.55,A -85,B 0,C 180,E1 -18108.574,E2 -18108.574} C_VEL
LIN {X 0,Y 266.862,Z 662.122,A -85,B 0,C 180,E1 -18111.229,E2 -18111.229} C_VEL
LIN {X 0,Y 269.208,Z 652.842,A -85,B 0,C 180,E1 -18113.642,E2 -18113.642} C_VEL
LIN {X 0,Y 271.942,Z 641.573,A -85,B 0,C 180,E1 -18116.061,E2 -18116.061} C_VEL
LIN {X 0,Y 274.954,Z 629.193,A -85,B 0,C 180,E1 -18118.219,E2 -18118.219} C_VEL
LIN {X 0,Y 277.851,Z 616.869,A -85,B 0,C 180,E1 -18119.969,E2 -18119.969} C_VEL
LIN {X 0,Y 279.013,Z 610.317,A -85,B 0,C 180,E1 -18120.791,E2 -18120.791} C_VEL
LIN {X 0,Y 277.817,Z 595.681,A -85,B 0,C 180,E1 -18122.712,E2 -18122.712} C_VEL
LIN {X 0,Y 275.77,Z 581.727,A -85,B 0,C 180,E1 -18124.334,E2 -18124.334} C_VEL
LIN {X 0,Y 272.51,Z 565.769,A -85,B 0,C 180,E1 -18125.987,E2 -18125.987} C_VEL
LIN {X 0,Y 268.09,Z 549.743,A -85,B 0,C 180,E1 -18127.488,E2 -18127.488} C_VEL
LIN {X 0,Y 265.164,Z 540.351,A -85,B 0,C 180,E1 -18128.277,E2 -18128.277} C_VEL
LIN {X 0,Y 265.128,Z 539.863,A -85,B 0,C 180,E1 -18128.341,E2 -18128.341} C_VEL
LIN {X 0,Y 265.992,Z 534.928,A -85,B 0,C 180,E1 -18132.285,E2 -18132.285} C_VEL
LIN {X 0,Y 266.021,Z 532.348,A -85,B 0,C 180,E1 -18134.496,E2 -18134.496} C_VEL
LIN {X 0,Y 265.194,Z 527.925,A -85,B 0,C 180,E1 -18138.507,E2 -18138.507} C_VEL
LIN {X 0,Y 264.324,Z 523.399,A -85,B 0,C 180,E1 -18142.904,E2 -18142.904} C_VEL
LIN {X 0,Y 263.856,Z 520.408,A -85,B 0,C 180,E1 -18145.99,E2 -18145.99} C_VEL
LIN {X 0,Y 263.344,Z 517.186,A -85,B 0,C 180,E1 -18149.532,E2 -18149.532} C_VEL
LIN {X 0,Y 263.182,Z 516.325,A -85,B 0,C 180,E1 -18150.615,E2 -18150.615} C_VEL
LIN {X 0,Y 263.185,Z 516.326,A -85,B 0,C 180,E1 -18154.707,E2 -18154.707} C_VEL
LIN {X 0,Y 263.255,Z 516.321,A -85,B 0,C 180,E1 -18159.693,E2 -18159.693} C_VEL
LIN {X 0,Y 263.343,Z 516.305,A -85,B 0,C 180,E1 -18164.522,E2 -18164.522} C_VEL
LIN {X 0,Y 263.366,Z 516.295,A -85,B 0,C 180,E1 -18169.235,E2 -18169.235} C_VEL
LIN {X 0,Y 263.564,Z 516.27,A -85,B 0,C 180,E1 -18172.339,E2 -18172.339} C_VEL
LIN {X 0,Y 263.747,Z 516.249,A -85,B 0,C 180,E1 -18178.474,E2 -18178.474} C_VEL
LIN {X 0,Y 263.745,Z 516.239,A -85,B 0,C 180,E1 -18181.528,E2 -18181.528} C_VEL
LIN {X 0,Y 263.552,Z 516.28,A -85,B 0,C 180,E1 -18187.663,E2 -18187.663} C_VEL
LIN {X 0,Y 263.348,Z 516.293,A -85,B 0,C 180,E1 -18190.767,E2 -18190.767} C_VEL
LIN {X 0,Y 263.338,Z 516.301,A -85,B 0,C 180,E1 -18195.479,E2 -18195.479} C_VEL
LIN {X 0,Y 263.257,Z 516.311,A -85,B 0,C 180,E1 -18200.308,E2 -18200.308} C_VEL
LIN {X 0,Y 263.203,Z 516.306,A -85,B 0,C 180,E1 -18205.293,E2 -18205.293} C_VEL
LIN {X 0,Y 263.171,Z 516.325,A -85,B 0,C 180,E1 -18208.731,E2 -18208.731} C_VEL
LIN {X 0,Y 263.13,Z 516.327,A -85,B 0,C 180,E1 -18212.29,E2 -18212.29} C_VEL
LIN {X 0,Y 263.186,Z 516.308,A -85,B 0,C 180,E1 -18215.979,E2 -18215.979} C_VEL
LIN {X 0,Y 263.16,Z 516.33,A -85,B 0,C 180,E1 -18219.864,E2 -18219.864} C_VEL
LIN {X 0,Y 263.189,Z 516.319,A -85,B 0,C 180,E1 -18223.866,E2 -18223.866} C_VEL
LIN {X 0,Y 263.193,Z 516.321,A -85,B 0,C 180,E1 -18228.122,E2 -18228.122} C_VEL
LIN {X 0,Y 263.188,Z 516.326,A -85,B 0,C 180,E1 -18232.11,E2 -18232.11} C_VEL
LIN {X 0,Y 263.184,Z 516.317,A -85,B 0,C 180,E1 -18235.892,E2 -18235.892} C_VEL
LIN {X 0,Y 263.152,Z 516.335,A -85,B 0,C 180,E1 -18239.509,E2 -18239.509} C_VEL
LIN {X 0,Y 263.196,Z 516.319,A -85,B 0,C 180,E1 -18243.004,E2 -18243.004} C_VEL
LIN {X 0,Y 263.192,Z 516.325,A -85,B 0,C 180,E1 -18246.389,E2 -18246.389} C_VEL
LIN {X 0,Y 263.266,Z 516.309,A -85,B 0,C 180,E1 -18249.695,E2 -18249.695} C_VEL
LIN {X 0,Y 263.354,Z 516.301,A -85,B 0,C 180,E1 -18254.523,E2 -18254.523} C_VEL
LIN {X 0,Y 263.359,Z 516.305,A -85,B 0,C 180,E1 -18259.235,E2 -18259.235} C_VEL
LIN {X 0,Y 263.549,Z 516.281,A -85,B 0,C 180,E1 -18262.339,E2 -18262.339} C_VEL
LIN {X 0,Y 263.757,Z 516.255,A -85,B 0,C 180,E1 -18268.474,E2 -18268.474} C_VEL
LIN {X 0,Y 263.618,Z 516.272,A -85,B 0,C 180,E1 -18271.528,E2 -18271.528} C_VEL
LIN {X 0,Y 263.566,Z 516.28,A -85,B 0,C 180,E1 -18271.73,E2 -18271.73} C_VEL
LIN {X 0,Y 264.555,Z 519.276,A -85,B 0,C 180,E1 -18272.023,E2 -18272.023} C_VEL
LIN {X 0,Y 271.594,Z 533.497,A -85,B 0,C 180,E1 -18273.787,E2 -18273.787} C_VEL
LIN {X 0,Y 275.106,Z 542.769,A -85,B 0,C 180,E1 -18274.913,E2 -18274.913} C_VEL
LIN {X 0,Y 279.542,Z 557.338,A -85,B 0,C 180,E1 -18276.762,E2 -18276.762} C_VEL
LIN {X 0,Y 282.304,Z 569.106,A -85,B 0,C 180,E1 -18278.374,E2 -18278.374} C_VEL
LIN {X 0,Y 282.547,Z 570.653,A -85,B 0,C 180,E1 -18278.584,E2 -18278.584} C_VEL
LIN {X 0,Y 279.987,Z 584.118,A -85,B 0,C 180,E1 -18280.12,E2 -18280.12} C_VEL
LIN {X 0,Y 277.249,Z 596.725,A -85,B 0,C 180,E1 -18281.886,E2 -18281.886} C_VEL
LIN {X 0,Y 274.607,Z 608.151,A -85,B 0,C 180,E1 -18283.837,E2 -18283.837} C_VEL
LIN {X 0,Y 271.727,Z 619.381,A -85,B 0,C 180,E1 -18286.144,E2 -18286.144} C_VEL
LIN {X 0,Y 269.25,Z 628.989,A -85,B 0,C 180,E1 -18288.547,E2 -18288.547} C_VEL
LIN {X 0,Y 266.951,Z 637.803,A -85,B 0,C 180,E1 -18291.223,E2 -18291.223} C_VEL
LIN {X 0,Y 264.907,Z 645.944,A -85,B 0,C 180,E1 -18294.282,E2 -18294.282} C_VEL
LIN {X 0,Y 263.549,Z 651.655,A -85,B 0,C 180,E1 -18296.958,E2 -18296.958} C_VEL
LIN {X 0,Y 262.587,Z 656.323,A -85,B 0,C 180,E1 -18299.679,E2 -18299.679} C_VEL
LIN {X 0,Y 261.821,Z 659.981,A -85,B 0,C 180,E1 -18302.47,E2 -18302.47} C_VEL
LIN {X 0,Y 261.435,Z 661.911,A -85,B 0,C 180,E1 -18304.37,E2 -18304.37} C_VEL
LIN {X 0,Y 261.145,Z 663.39,A -85,B 0,C 180,E1 -18306.304,E2 -18306.304} C_VEL
LIN {X 0,Y 261.003,Z 664.544,A -85,B 0,C 180,E1 -18308.658,E2 -18308.658} C_VEL
LIN {X 0,Y 261.052,Z 665.098,A -85,B 0,C 180,E1 -18311.077,E2 -18311.077} C_VEL
LIN {X 0,Y 261.325,Z 664.706,A -85,B 0,C 180,E1 -18314.366,E2 -18314.366} C_VEL
LIN {X 0,Y 261.712,Z 663.816,A -85,B 0,C 180,E1 -18316.473,E2 -18316.473} C_VEL
LIN {X 0,Y 262.771,Z 661.004,A -85,B 0,C 180,E1 -18320.066,E2 -18320.066} C_VEL
LIN {X 0,Y 264.008,Z 657.498,A -85,B 0,C 180,E1 -18322.998,E2 -18322.998} C_VEL
LIN {X 0,Y 266.005,Z 652.114,A -85,B 0,C 180,E1 -18326.3,E2 -18326.3} C_VEL
LIN {X 0,Y 268.753,Z 644.841,A -85,B 0,C 180,E1 -18329.651,E2 -18329.651} C_VEL
LIN {X 0,Y 271.388,Z 637.807,A -85,B 0,C 180,E1 -18332.215,E2 -18332.215} C_VEL
LIN {X 0,Y 274.293,Z 629.871,A -85,B 0,C 180,E1 -18334.584,E2 -18334.584} C_VEL
LIN {X 0,Y 277.719,Z 620.116,A -85,B 0,C 180,E1 -18336.992,E2 -18336.992} C_VEL
LIN {X 0,Y 280.903,Z 610.551,A -85,B 0,C 180,E1 -18338.951,E2 -18338.951} C_VEL
LIN {X 0,Y 284.329,Z 599.365,A -85,B 0,C 180,E1 -18340.86,E2 -18340.86} C_VEL
LIN {X 0,Y 287.878,Z 586.55,A -85,B 0,C 180,E1 -18342.643,E2 -18342.643} C_VEL
LIN {X 0,Y 289.891,Z 578.184,A -85,B 0,C 180,E1 -18343.63,E2 -18343.63} C_VEL
LIN {X 0,Y 288.788,Z 571.276,A -85,B 0,C 180,E1 -18344.834,E2 -18344.834} C_VEL
LIN {X 0,Y 285.749,Z 560.116,A -85,B 0,C 180,E1 -18346.882,E2 -18346.882} C_VEL
LIN {X 0,Y 281.448,Z 548.612,A -85,B 0,C 180,E1 -18349.118,E2 -18349.118} C_VEL
LIN {X 0,Y 275.867,Z 537.643,A -85,B 0,C 180,E1 -18351.522,E2 -18351.522} C_VEL
LIN {X 0,Y 273.233,Z 533.173,A -85,B 0,C 180,E1 -18352.61,E2 -18352.61} C_VEL
LIN {X 0,Y 270.629,Z 529.174,A -85,B 0,C 180,E1 -18353.663,E2 -18353.663} C_VEL
LIN {X 0,Y 268.363,Z 526.108,A -85,B 0,C 180,E1 -18354.576,E2 -18354.576} C_VEL
LIN {X 0,Y 267.697,Z 524.739,A -85,B 0,C 180,E1 -18354.873,E2 -18354.873} C_VEL
LIN {X 0,Y 265.426,Z 522.739,A -85,B 0,C 180,E1 -18355.729,E2 -18355.729} C_VEL
LIN {X 0,Y 264.187,Z 520.241,A -85,B 0,C 180,E1 -18356.329,E2 -18356.329} C_VEL
LIN {X 0,Y 264,Z 519.453,A -85,B 0,C 180,E1 -18356.47,E2 -18356.47} C_VEL
LIN {X 0,Y 264.22,Z 518.661,A -85,B 0,C 180,E1 -18359.999,E2 -18359.999} C_VEL
LIN {X 0,Y 263.92,Z 518.267,A -85,B 0,C 180,E1 -18363.052,E2 -18363.052} C_VEL
LIN {X 0,Y 263.734,Z 518.081,A -85,B 0,C 180,E1 -18365.385,E2 -18365.385} C_VEL
LIN {X 0,Y 263.117,Z 518.152,A -85,B 0,C 180,E1 -18366.661,E2 -18366.661} C_VEL
LIN {X 0,Y 260.279,Z 518.757,A -85,B 0,C 180,E1 -18368.74,E2 -18368.74} C_VEL
LIN {X 0,Y 257.849,Z 519.352,A -85,B 0,C 180,E1 -18370.43,E2 -18370.43} C_VEL
LIN {X 0,Y 256.818,Z 519.667,A -85,B 0,C 180,E1 -18371.742,E2 -18371.742} C_VEL
LIN {X 0,Y 256.743,Z 519.722,A -85,B 0,C 180,E1 -18372.187,E2 -18372.187} C_VEL
LIN {X 0,Y 256.825,Z 520.346,A -85,B 0,C 180,E1 -18376.711,E2 -18376.711} C_VEL
LIN {X 0,Y 256.911,Z 521.381,A -85,B 0,C 180,E1 -18380.831,E2 -18380.831} C_VEL
LIN {X 0,Y 257.2,Z 523.078,A -85,B 0,C 180,E1 -18385.615,E2 -18385.615} C_VEL
LIN {X 0,Y 257.453,Z 524.888,A -85,B 0,C 180,E1 -18389.43,E2 -18389.43} C_VEL
LIN {X 0,Y 257.768,Z 526.952,A -85,B 0,C 180,E1 -18393.044,E2 -18393.044} C_VEL
LIN {X 0,Y 258.237,Z 529.434,A -85,B 0,C 180,E1 -18396.779,E2 -18396.779} C_VEL
LIN {X 0,Y 258.786,Z 532.865,A -85,B 0,C 180,E1 -18401.19,E2 -18401.19} C_VEL
LIN {X 0,Y 258.866,Z 533.304,A -85,B 0,C 180,E1 -18401.694,E2 -18401.694} C_VEL
LIN {X 0,Y 259.901,Z 536.301,A -85,B 0,C 180,E1 -18402.271,E2 -18402.271} C_VEL
LIN {X 0,Y 262.331,Z 539.565,A -85,B 0,C 180,E1 -18403.354,E2 -18403.354} C_VEL
LIN {X 0,Y 262.932,Z 540.633,A -85,B 0,C 180,E1 -18403.626,E2 -18403.626} C_VEL
LIN {X 0,Y 264.576,Z 544.068,A -85,B 0,C 180,E1 -18404.381,E2 -18404.381} C_VEL
LIN {X 0,Y 266.199,Z 546.528,A -85,B 0,C 180,E1 -18405.072,E2 -18405.072} C_VEL
LIN {X 0,Y 268.61,Z 552.061,A -85,B 0,C 180,E1 -18406.217,E2 -18406.217} C_VEL
LIN {X 0,Y 271.608,Z 560.083,A -85,B 0,C 180,E1 -18407.719,E2 -18407.719} C_VEL
LIN {X 0,Y 275.322,Z 573.409,A -85,B 0,C 180,E1 -18409.977,E2 -18409.977} C_VEL
LIN {X 0,Y 277.411,Z 584.742,A -85,B 0,C 180,E1 -18411.753,E2 -18411.753} C_VEL
LIN {X 0,Y 278.589,Z 596.272,A -85,B 0,C 180,E1 -18413.532,E2 -18413.532} C_VEL
LIN {X 0,Y 278.794,Z 608.56,A -85,B 0,C 180,E1 -18415.445,E2 -18415.445} C_VEL
LIN {X 0,Y 278.412,Z 615.419,A -85,B 0,C 180,E1 -18416.545,E2 -18416.545} C_VEL
LIN {X 0,Y 274.687,Z 627.984,A -85,B 0,C 180,E1 -18418.365,E2 -18418.365} C_VEL
LIN {X 0,Y 270.765,Z 639.841,A -85,B 0,C 180,E1 -18420.451,E2 -18420.451} C_VEL
LIN {X 0,Y 267.262,Z 649.935,A -85,B 0,C 180,E1 -18422.601,E2 -18422.601} C_VEL
LIN {X 0,Y 263.735,Z 659.914,A -85,B 0,C 180,E1 -18425.189,E2 -18425.189} C_VEL
LIN {X 0,Y 260.864,Z 668.291,A -85,B 0,C 180,E1 -18427.841,E2 -18427.841} C_VEL
LIN {X 0,Y 258.229,Z 676.258,A -85,B 0,C 180,E1 -18430.937,E2 -18430.937} C_VEL
LIN {X 0,Y 256.199,Z 682.678,A -85,B 0,C 180,E1 -18434.078,E2 -18434.078} C_VEL
LIN {X 0,Y 254.998,Z 687.742,A -85,B 0,C 180,E1 -18437.262,E2 -18437.262} C_VEL
LIN {X 0,Y 254.299,Z 691.541,A -85,B 0,C 180,E1 -18440.454,E2 -18440.454} C_VEL
LIN {X 0,Y 254.134,Z 694.14,A -85,B 0,C 180,E1 -18443.648,E2 -18443.648} C_VEL
LIN {X 0,Y 254.209,Z 695.567,A -85,B 0,C 180,E1 -18446.83,E2 -18446.83} C_VEL
LIN {X 0,Y 254.354,Z 695.763,A -85,B 0,C 180,E1 -18449.999,E2 -18449.999} C_VEL
LIN {X 0,Y 254.236,Z 694.738,A -85,B 0,C 180,E1 -18453.168,E2 -18453.168} C_VEL
LIN {X 0,Y 254.244,Z 692.496,A -85,B 0,C 180,E1 -18456.347,E2 -18456.347} C_VEL
LIN {X 0,Y 254.338,Z 688.974,A -85,B 0,C 180,E1 -18459.542,E2 -18459.542} C_VEL
LIN {X 0,Y 254.967,Z 684.111,A -85,B 0,C 180,E1 -18462.738,E2 -18462.738} C_VEL
LIN {X 0,Y 256.108,Z 677.768,A -85,B 0,C 180,E1 -18465.926,E2 -18465.926} C_VEL
LIN {X 0,Y 257.661,Z 670.912,A -85,B 0,C 180,E1 -18468.692,E2 -18468.692} C_VEL
LIN {X 0,Y 259.795,Z 662.608,A -85,B 0,C 180,E1 -18471.419,E2 -18471.419} C_VEL
LIN {X 0,Y 262.389,Z 652.794,A -85,B 0,C 180,E1 -18474.062,E2 -18474.062} C_VEL
LIN {X 0,Y 264.997,Z 642.4,A -85,B 0,C 180,E1 -18476.373,E2 -18476.373} C_VEL
LIN {X 0,Y 268.117,Z 630.295,A -85,B 0,C 180,E1 -18478.578,E2 -18478.578} C_VEL
LIN {X 0,Y 271.032,Z 618.224,A -85,B 0,C 180,E1 -18480.373,E2 -18480.373} C_VEL
LIN {X 0,Y 272.232,Z 612.717,A -85,B 0,C 180,E1 -18481.084,E2 -18481.084} C_VEL
LIN {X 0,Y 271.928,Z 604.425,A -85,B 0,C 180,E1 -18482.249,E2 -18482.249} C_VEL
LIN {X 0,Y 270.681,Z 592.402,A -85,B 0,C 180,E1 -18483.815,E2 -18483.815} C_VEL
LIN {X 0,Y 268.505,Z 578.604,A -85,B 0,C 180,E1 -18485.445,E2 -18485.445} C_VEL
LIN {X 0,Y 265.352,Z 563.788,A -85,B 0,C 180,E1 -18487.021,E2 -18487.021} C_VEL
LIN {X 0,Y 261.311,Z 549.465,A -85,B 0,C 180,E1 -18488.415,E2 -18488.415} C_VEL
LIN {X 0,Y 258.369,Z 540.398,A -85,B 0,C 180,E1 -18489.228,E2 -18489.228} C_VEL
LIN {X 0,Y 258.262,Z 539.473,A -85,B 0,C 180,E1 -18489.312,E2 -18489.312} C_VEL
LIN {X 0,Y 258.992,Z 535.19,A -85,B 0,C 180,E1 -18492.89,E2 -18492.89} C_VEL
LIN {X 0,Y 258.87,Z 532.632,A -85,B 0,C 180,E1 -18495.101,E2 -18495.101} C_VEL
LIN {X 0,Y 258.019,Z 528.312,A -85,B 0,C 180,E1 -18499.178,E2 -18499.178} C_VEL
LIN {X 0,Y 257.301,Z 524.441,A -85,B 0,C 180,E1 -18503.065,E2 -18503.065} C_VEL
LIN {X 0,Y 256.734,Z 520.944,A -85,B 0,C 180,E1 -18506.805,E2 -18506.805} C_VEL
LIN {X 0,Y 256.197,Z 517.395,A -85,B 0,C 180,E1 -18510.843,E2 -18510.843} C_VEL
LIN {X 0,Y 256.135,Z 517.206,A -85,B 0,C 180,E1 -18515.696,E2 -18515.696} C_VEL
LIN {X 0,Y 256.154,Z 517.204,A -85,B 0,C 180,E1 -18519.104,E2 -18519.104} C_VEL
LIN {X 0,Y 256.292,Z 517.185,A -85,B 0,C 180,E1 -18524.085,E2 -18524.085} C_VEL
LIN {X 0,Y 256.302,Z 517.178,A -85,B 0,C 180,E1 -18528.934,E2 -18528.934} C_VEL
LIN {X 0,Y 256.532,Z 517.145,A -85,B 0,C 180,E1 -18532.127,E2 -18532.127} C_VEL
LIN {X 0,Y 256.71,Z 517.125,A -85,B 0,C 180,E1 -18538.432,E2 -18538.432} C_VEL
LIN {X 0,Y 256.708,Z 517.114,A -85,B 0,C 180,E1 -18541.569,E2 -18541.569} C_VEL
LIN {X 0,Y 256.466,Z 517.159,A -85,B 0,C 180,E1 -18546.72,E2 -18546.72} C_VEL
LIN {X 0,Y 256.42,Z 517.161,A -85,B 0,C 180,E1 -18549.466,E2 -18549.466} C_VEL
LIN {X 0,Y 256.244,Z 517.18,A -85,B 0,C 180,E1 -18554.291,E2 -18554.291} C_VEL
LIN {X 0,Y 256.203,Z 517.197,A -85,B 0,C 180,E1 -18557.563,E2 -18557.563} C_VEL
LIN {X 0,Y 256.152,Z 517.196,A -85,B 0,C 180,E1 -18561.121,E2 -18561.121} C_VEL
LIN {X 0,Y 256.183,Z 517.178,A -85,B 0,C 180,E1 -18565.14,E2 -18565.14} C_VEL
LIN {X 0,Y 256.107,Z 517.21,A -85,B 0,C 180,E1 -18569.601,E2 -18569.601} C_VEL
LIN {X 0,Y 256.081,Z 517.202,A -85,B 0,C 180,E1 -18573.292,E2 -18573.292} C_VEL
LIN {X 0,Y 256.138,Z 517.189,A -85,B 0,C 180,E1 -18577.28,E2 -18577.28} C_VEL
LIN {X 0,Y 256.13,Z 517.206,A -85,B 0,C 180,E1 -18581.19,E2 -18581.19} C_VEL
LIN {X 0,Y 256.115,Z 517.191,A -85,B 0,C 180,E1 -18585.518,E2 -18585.518} C_VEL
LIN {X 0,Y 256.121,Z 517.202,A -85,B 0,C 180,E1 -18588.812,E2 -18588.812} C_VEL
LIN {X 0,Y 256.155,Z 517.202,A -85,B 0,C 180,E1 -18592.873,E2 -18592.873} C_VEL
LIN {X 0,Y 256.085,Z 517.203,A -85,B 0,C 180,E1 -18596.712,E2 -18596.712} C_VEL
LIN {X 0,Y 256.139,Z 517.205,A -85,B 0,C 180,E1 -18601.406,E2 -18601.406} C_VEL
LIN {X 0,Y 256.174,Z 517.199,A -85,B 0,C 180,E1 -18605.701,E2 -18605.701} C_VEL
LIN {X 0,Y 256.17,Z 517.197,A -85,B 0,C 180,E1 -18609.106,E2 -18609.106} C_VEL
LIN {X 0,Y 256.303,Z 517.181,A -85,B 0,C 180,E1 -18614.086,E2 -18614.086} C_VEL
LIN {X 0,Y 256.299,Z 517.183,A -85,B 0,C 180,E1 -18617.329,E2 -18617.329} C_VEL
LIN {X 0,Y 256.509,Z 517.159,A -85,B 0,C 180,E1 -18622.127,E2 -18622.127} C_VEL
LIN {X 0,Y 256.505,Z 517.158,A -85,B 0,C 180,E1 -18626.86,E2 -18626.86} C_VEL
LIN {X 0,Y 256.747,Z 517.127,A -85,B 0,C 180,E1 -18630.001,E2 -18630.001} C_VEL
LIN {X 0,Y 256.638,Z 517.138,A -85,B 0,C 180,E1 -18630.736,E2 -18630.736} C_VEL
LIN {X 0,Y 257.751,Z 520.197,A -85,B 0,C 180,E1 -18631.075,E2 -18631.075} C_VEL
LIN {X 0,Y 265.15,Z 535.314,A -85,B 0,C 180,E1 -18633.039,E2 -18633.039} C_VEL
LIN {X 0,Y 268.084,Z 542.544,A -85,B 0,C 180,E1 -18633.979,E2 -18633.979} C_VEL
LIN {X 0,Y 272.603,Z 557.276,A -85,B 0,C 180,E1 -18635.92,E2 -18635.92} C_VEL
LIN {X 0,Y 275.334,Z 568.552,A -85,B 0,C 180,E1 -18637.517,E2 -18637.517} C_VEL
LIN {X 0,Y 276.008,Z 572.299,A -85,B 0,C 180,E1 -18638.051,E2 -18638.051} C_VEL
LIN {X 0,Y 273.383,Z 585.544,A -85,B 0,C 180,E1 -18639.62,E2 -18639.62} C_VEL
LIN {X 0,Y 270.541,Z 598.161,A -85,B 0,C 180,E1 -18641.453,E2 -18641.453} C_VEL
LIN {X 0,Y 267.501,Z 610.639,A -85,B 0,C 180,E1 -18643.678,E2 -18643.678} C_VEL
LIN {X 0,Y 264.534,Z 621.871,A -85,B 0,C 180,E1 -18646.132,E2 -18646.132} C_VEL
LIN {X 0,Y 261.852,Z 631.807,A -85,B 0,C 180,E1 -18648.789,E2 -18648.789} C_VEL
LIN {X 0,Y 259.647,Z 639.939,A -85,B 0,C 180,E1 -18651.433,E2 -18651.433} C_VEL
LIN {X 0,Y 257.886,Z 646.711,A -85,B 0,C 180,E1 -18654.129,E2 -18654.129} C_VEL
LIN {X 0,Y 256.492,Z 652.356,A -85,B 0,C 180,E1 -18656.879,E2 -18656.879} C_VEL
LIN {X 0,Y 255.504,Z 656.961,A -85,B 0,C 180,E1 -18659.678,E2 -18659.678} C_VEL
LIN {X 0,Y 254.718,Z 660.594,A -85,B 0,C 180,E1 -18662.55,E2 -18662.55} C_VEL
LIN {X 0,Y 254.157,Z 663.226,A -85,B 0,C 180,E1 -18665.5,E2 -18665.5} C_VEL
LIN {X 0,Y 253.969,Z 664.459,A -85,B 0,C 180,E1 -18667.503,E2 -18667.503} C_VEL
LIN {X 0,Y 253.908,Z 665.254,A -85,B 0,C 180,E1 -18669.541,E2 -18669.541} C_VEL
LIN {X 0,Y 254.006,Z 665.563,A -85,B 0,C 180,E1 -18671.663,E2 -18671.663} C_VEL
LIN {X 0,Y 254.204,Z 665.29,A -85,B 0,C 180,E1 -18674.041,E2 -18674.041} C_VEL
LIN {X 0,Y 254.593,Z 664.456,A -85,B 0,C 180,E1 -18676.359,E2 -18676.359} C_VEL
LIN {X 0,Y 255.206,Z 663.059,A -85,B 0,C 180,E1 -18678.629,E2 -18678.629} C_VEL
LIN {X 0,Y 255.982,Z 661.066,A -85,B 0,C 180,E1 -18680.841,E2 -18680.841} C_VEL
LIN {X 0,Y 257.446,Z 657.258,A -85,B 0,C 180,E1 -18683.989,E2 -18683.989} C_VEL
LIN {X 0,Y 259.567,Z 651.95,A -85,B 0,C 180,E1 -18687.212,E2 -18687.212} C_VEL
LIN {X 0,Y 262.269,Z 645.252,A -85,B 0,C 180,E1 -18690.329,E2 -18690.329} C_VEL
LIN {X 0,Y 265.414,Z 637.311,A -85,B 0,C 180,E1 -18693.246,E2 -18693.246} C_VEL
LIN {X 0,Y 268.619,Z 629.088,A -85,B 0,C 180,E1 -18695.706,E2 -18695.706} C_VEL
LIN {X 0,Y 272.428,Z 618.728,A -85,B 0,C 180,E1 -18698.235,E2 -18698.235} C_VEL
LIN {X 0,Y 276.434,Z 606.932,A -85,B 0,C 180,E1 -18700.557,E2 -18700.557} C_VEL
LIN {X 0,Y 280.444,Z 593.78,A -85,B 0,C 180,E1 -18702.642,E2 -18702.642} C_VEL
LIN {X 0,Y 283.671,Z 581.928,A -85,B 0,C 180,E1 -18704.185,E2 -18704.185} C_VEL
LIN {X 0,Y 284.127,Z 580.062,A -85,B 0,C 180,E1 -18704.395,E2 -18704.395} C_VEL
LIN {X 0,Y 282.586,Z 571.535,A -85,B 0,C 180,E1 -18706.003,E2 -18706.003} C_VEL
LIN {X 0,Y 279.128,Z 559.482,A -85,B 0,C 180,E1 -18708.379,E2 -18708.379} C_VEL
LIN {X 0,Y 275.69,Z 550.589,A -85,B 0,C 180,E1 -18710.252,E2 -18710.252} C_VEL
LIN {X 0,Y 270.076,Z 539.45,A -85,B 0,C 180,E1 -18712.911,E2 -18712.911} C_VEL
LIN {X 0,Y 267.207,Z 534.933,A -85,B 0,C 180,E1 -18714.207,E2 -18714.207} C_VEL
LIN {X 0,Y 264.642,Z 530.987,A -85,B 0,C 180,E1 -18715.347,E2 -18715.347} C_VEL
LIN {X 0,Y 262.061,Z 527.992,A -85,B 0,C 180,E1 -18716.492,E2 -18716.492} C_VEL
LIN {X 0,Y 260.808,Z 525.606,A -85,B 0,C 180,E1 -18717.118,E2 -18717.118} C_VEL
LIN {X 0,Y 258.526,Z 523.44,A -85,B 0,C 180,E1 -18718.131,E2 -18718.131} C_VEL
LIN {X 0,Y 257.313,Z 520.779,A -85,B 0,C 180,E1 -18718.826,E2 -18718.826} C_VEL
LIN {X 0,Y 257.234,Z 520.326,A -85,B 0,C 180,E1 -18719.021,E2 -18719.021} C_VEL
LIN {X 0,Y 257.137,Z 519.935,A -85,B 0,C 180,E1 -18721.566,E2 -18721.566} C_VEL
LIN {X 0,Y 256.874,Z 519.561,A -85,B 0,C 180,E1 -18726.282,E2 -18726.282} C_VEL
LIN {X 0,Y 256.851,Z 519.55,A -85,B 0,C 180,E1 -18729.926,E2 -18729.926} C_VEL
LIN {X 0,Y 256.743,Z 519.722,A -85,B 0,C 180,E1 -18732.187,E2 -18732.187} C_VEL
LIN {X 0,Y 256.106,Z 520.012,A -85,B 0,C 180,E1 -18733.497,E2 -18733.497} C_VEL
LIN {X 0,Y 253.304,Z 520.983,A -85,B 0,C 180,E1 -18735.627,E2 -18735.627} C_VEL
LIN {X 0,Y 250.938,Z 521.87,A -85,B 0,C 180,E1 -18737.359,E2 -18737.359} C_VEL
LIN {X 0,Y 249.96,Z 522.408,A -85,B 0,C 180,E1 -18738.704,E2 -18738.704} C_VEL
LIN {X 0,Y 249.901,Z 522.537,A -85,B 0,C 180,E1 -18739.159,E2 -18739.159} C_VEL
LIN {X 0,Y 250.066,Z 523.757,A -85,B 0,C 180,E1 -18743.17,E2 -18743.17} C_VEL
LIN {X 0,Y 250.338,Z 525.147,A -85,B 0,C 180,E1 -18746.691,E2 -18746.691} C_VEL
LIN {X 0,Y 250.581,Z 526.931,A -85,B 0,C 180,E1 -18750.32,E2 -18750.32} C_VEL
LIN {X 0,Y 250.947,Z 529.103,A -85,B 0,C 180,E1 -18754.063,E2 -18754.063} C_VEL
LIN {X 0,Y 251.461,Z 531.725,A -85,B 0,C 180,E1 -18757.942,E2 -18757.942} C_VEL
LIN {X 0,Y 251.517,Z 532.249,A -85,B 0,C 180,E1 -18758.625,E2 -18758.625} C_VEL
LIN {X 0,Y 252.689,Z 535.494,A -85,B 0,C 180,E1 -18759.404,E2 -18759.404} C_VEL
LIN {X 0,Y 255.339,Z 538.84,A -85,B 0,C 180,E1 -18760.791,E2 -18760.791} C_VEL
LIN {X 0,Y 255.892,Z 539.691,A -85,B 0,C 180,E1 -18761.069,E2 -18761.069} C_VEL
LIN {X 0,Y 257.733,Z 543.47,A -85,B 0,C 180,E1 -18762.05,E2 -18762.05} C_VEL
LIN {X 0,Y 259.449,Z 545.928,A -85,B 0,C 180,E1 -18762.882,E2 -18762.882} C_VEL
LIN {X 0,Y 261.508,Z 550.227,A -85,B 0,C 180,E1 -18763.951,E2 -18763.951} C_VEL
LIN {X 0,Y 262.564,Z 552.001,A -85,B 0,C 180,E1 -18764.436,E2 -18764.436} C_VEL
LIN {X 0,Y 264.769,Z 557.546,A -85,B 0,C 180,E1 -18765.645,E2 -18765.645} C_VEL
LIN {X 0,Y 267.949,Z 567.359,A -85,B 0,C 180,E1 -18767.541,E2 -18767.541} C_VEL
LIN {X 0,Y 270.702,Z 579.452,A -85,B 0,C 180,E1 -18769.667,E2 -18769.667} C_VEL
LIN {X 0,Y 272.201,Z 589.697,A -85,B 0,C 180,E1 -18771.354,E2 -18771.354} C_VEL
LIN {X 0,Y 272.94,Z 601.405,A -85,B 0,C 180,E1 -18773.267,E2 -18773.267} C_VEL
LIN {X 0,Y 272.693,Z 613.368,A -85,B 0,C 180,E1 -18775.234,E2 -18775.234} C_VEL
LIN {X 0,Y 272.308,Z 617.137,A -85,B 0,C 180,E1 -18775.87,E2 -18775.87} C_VEL
LIN {X 0,Y 268.329,Z 629.497,A -85,B 0,C 180,E1 -18777.747,E2 -18777.747} C_VEL
LIN {X 0,Y 263.969,Z 641.899,A -85,B 0,C 180,E1 -18780.052,E2 -18780.052} C_VEL
LIN {X 0,Y 259.813,Z 653.081,A -85,B 0,C 180,E1 -18782.622,E2 -18782.622} C_VEL
LIN {X 0,Y 256.347,Z 662.596,A -85,B 0,C 180,E1 -18785.337,E2 -18785.337} C_VEL
LIN {X 0,Y 253.424,Z 670.339,A -85,B 0,C 180,E1 -18788.013,E2 -18788.013} C_VEL
LIN {X 0,Y 250.86,Z 677.829,A -85,B 0,C 180,E1 -18791.205,E2 -18791.205} C_VEL
LIN {X 0,Y 248.937,Z 683.848,A -85,B 0,C 180,E1 -18794.442,E2 -18794.442} C_VEL
LIN {X 0,Y 247.737,Z 688.545,A -85,B 0,C 180,E1 -18797.715,E2 -18797.715} C_VEL
LIN {X 0,Y 247.248,Z 691.219,A -85,B 0,C 180,E1 -18800.18,E2 -18800.18} C_VEL
LIN {X 0,Y 247.037,Z 693.765,A -85,B 0,C 180,E1 -18803.465,E2 -18803.465} C_VEL
LIN {X 0,Y 247.115,Z 695.145,A -85,B 0,C 180,E1 -18806.738,E2 -18806.738} C_VEL
LIN {X 0,Y 247.269,Z 695.319,A -85,B 0,C 180,E1 -18809.999,E2 -18809.999} C_VEL
LIN {X 0,Y 247.168,Z 694.241,A -85,B 0,C 180,E1 -18813.259,E2 -18813.259} C_VEL
LIN {X 0,Y 247.157,Z 691.943,A -85,B 0,C 180,E1 -18816.53,E2 -18816.53} C_VEL
LIN {X 0,Y 247.287,Z 688.364,A -85,B 0,C 180,E1 -18819.817,E2 -18819.817} C_VEL
LIN {X 0,Y 247.954,Z 683.435,A -85,B 0,C 180,E1 -18823.105,E2 -18823.105} C_VEL
LIN {X 0,Y 249.308,Z 676.585,A -85,B 0,C 180,E1 -18826.574,E2 -18826.574} C_VEL
LIN {X 0,Y 251.137,Z 668.964,A -85,B 0,C 180,E1 -18829.621,E2 -18829.621} C_VEL
LIN {X 0,Y 253.485,Z 660.375,A -85,B 0,C 180,E1 -18832.408,E2 -18832.408} C_VEL
LIN {X 0,Y 256.128,Z 650.225,A -85,B 0,C 180,E1 -18835.11,E2 -18835.11} C_VEL
LIN {X 0,Y 259.06,Z 639.424,A -85,B 0,C 180,E1 -18837.463,E2 -18837.463} C_VEL
LIN {X 0,Y 262.02,Z 627.945,A -85,B 0,C 180,E1 -18839.527,E2 -18839.527} C_VEL
LIN {X 0,Y 265.177,Z 615.56,A -85,B 0,C 180,E1 -18841.339,E2 -18841.339} C_VEL
LIN {X 0,Y 265.652,Z 611.195,A -85,B 0,C 180,E1 -18841.944,E2 -18841.944} C_VEL
LIN {X 0,Y 264.642,Z 597.453,A -85,B 0,C 180,E1 -18843.894,E2 -18843.894} C_VEL
LIN {X 0,Y 262.763,Z 583.53,A -85,B 0,C 180,E1 -18845.668,E2 -18845.668} C_VEL
LIN {X 0,Y 259.884,Z 568.781,A -85,B 0,C 180,E1 -18847.354,E2 -18847.354} C_VEL
LIN {X 0,Y 256.117,Z 554.366,A -85,B 0,C 180,E1 -18848.866,E2 -18848.866} C_VEL
LIN {X 0,Y 251.57,Z 540.11,A -85,B 0,C 180,E1 -18850.255,E2 -18850.255} C_VEL
LIN {X 0,Y 251.441,Z 539.014,A -85,B 0,C 180,E1 -18850.398,E2 -18850.398} C_VEL
LIN {X 0,Y 251.98,Z 535.357,A -85,B 0,C 180,E1 -18853.518,E2 -18853.518} C_VEL
LIN {X 0,Y 251.559,Z 532.079,A -85,B 0,C 180,E1 -18856.582,E2 -18856.582} C_VEL
LIN {X 0,Y 250.877,Z 528.735,A -85,B 0,C 180,E1 -18859.886,E2 -18859.886} C_VEL
LIN {X 0,Y 250.071,Z 524.224,A -85,B 0,C 180,E1 -18864.586,E2 -18864.586} C_VEL
LIN {X 0,Y 249.635,Z 521.449,A -85,B 0,C 180,E1 -18867.663,E2 -18867.663} C_VEL
LIN {X 0,Y 249.085,Z 518.083,A -85,B 0,C 180,E1 -18871.797,E2 -18871.797} C_VEL
LIN {X 0,Y 249.127,Z 518.078,A -85,B 0,C 180,E1 -18874.967,E2 -18874.967} C_VEL
LIN {X 0,Y 249.101,Z 518.082,A -85,B 0,C 180,E1 -18880.211,E2 -18880.211} C_VEL
LIN {X 0,Y 249.235,Z 518.067,A -85,B 0,C 180,E1 -18883.622,E2 -18883.622} C_VEL
LIN {X 0,Y 249.246,Z 518.057,A -85,B 0,C 180,E1 -18888.617,E2 -18888.617} C_VEL
LIN {X 0,Y 249.474,Z 518.02,A -85,B 0,C 180,E1 -18891.903,E2 -18891.903} C_VEL
LIN {X 0,Y 249.435,Z 518.037,A -85,B 0,C 180,E1 -18896.77,E2 -18896.77} C_VEL
LIN {X 0,Y 249.721,Z 517.983,A -85,B 0,C 180,E1 -18900.001,E2 -18900.001} C_VEL
LIN {X 0,Y 249.432,Z 518.028,A -85,B 0,C 180,E1 -18903.231,E2 -18903.231} C_VEL
LIN {X 0,Y 249.436,Z 518.036,A -85,B 0,C 180,E1 -18906.704,E2 -18906.704} C_VEL
LIN {X 0,Y 249.336,Z 518.04,A -85,B 0,C 180,E1 -18909.737,E2 -18909.737} C_VEL
LIN {X 0,Y 249.194,Z 518.057,A -85,B 0,C 180,E1 -18914.705,E2 -18914.705} C_VEL
LIN {X 0,Y 249.133,Z 518.076,A -85,B 0,C 180,E1 -18918.079,E2 -18918.079} C_VEL
LIN {X 0,Y 249.082,Z 518.071,A -85,B 0,C 180,E1 -18921.519,E2 -18921.519} C_VEL
LIN {X 0,Y 249.126,Z 518.058,A -85,B 0,C 180,E1 -18925.483,E2 -18925.483} C_VEL
LIN {X 0,Y 249.076,Z 518.082,A -85,B 0,C 180,E1 -18928.994,E2 -18928.994} C_VEL
LIN {X 0,Y 249.032,Z 518.082,A -85,B 0,C 180,E1 -18932.426,E2 -18932.426} C_VEL
LIN {X 0,Y 249.072,Z 518.064,A -85,B 0,C 180,E1 -18936.339,E2 -18936.339} C_VEL
LIN {X 0,Y 249.081,Z 518.082,A -85,B 0,C 180,E1 -18940.464,E2 -18940.464} C_VEL
LIN {X 0,Y 249.092,Z 518.079,A -85,B 0,C 180,E1 -18942.815,E2 -18942.815} C_VEL
LIN {X 0,Y 249.089,Z 518.067,A -85,B 0,C 180,E1 -18947.38,E2 -18947.38} C_VEL
LIN {X 0,Y 249.052,Z 518.091,A -85,B 0,C 180,E1 -18951.626,E2 -18951.626} C_VEL
LIN {X 0,Y 249.061,Z 518.073,A -85,B 0,C 180,E1 -18955.644,E2 -18955.644} C_VEL
LIN {X 0,Y 249.053,Z 518.091,A -85,B 0,C 180,E1 -18959.475,E2 -18959.475} C_VEL
LIN {X 0,Y 249.077,Z 518.075,A -85,B 0,C 180,E1 -18963.164,E2 -18963.164} C_VEL
LIN {X 0,Y 249.085,Z 518.083,A -85,B 0,C 180,E1 -18966.735,E2 -18966.735} C_VEL
LIN {X 0,Y 249.113,Z 518.069,A -85,B 0,C 180,E1 -18970.213,E2 -18970.213} C_VEL
LIN {X 0,Y 249.245,Z 518.063,A -85,B 0,C 180,E1 -18973.623,E2 -18973.623} C_VEL
LIN {X 0,Y 249.248,Z 518.062,A -85,B 0,C 180,E1 -18978.617,E2 -18978.617} C_VEL
LIN {X 0,Y 249.45,Z 518.038,A -85,B 0,C 180,E1 -18981.903,E2 -18981.903} C_VEL
LIN {X 0,Y 249.301,Z 518.052,A -85,B 0,C 180,E1 -18985.149,E2 -18985.149} C_VEL
LIN {X 0,Y 249.686,Z 518.01,A -85,B 0,C 180,E1 -18989.194,E2 -18989.194} C_VEL
LIN {X 0,Y 249.7,Z 518.007,A -85,B 0,C 180,E1 -18989.698,E2 -18989.698} C_VEL
LIN {X 0,Y 250.823,Z 521.033,A -85,B 0,C 180,E1 -18990.051,E2 -18990.051} C_VEL
LIN {X 0,Y 254.874,Z 529.098,A -85,B 0,C 180,E1 -18991.136,E2 -18991.136} C_VEL
LIN {X 0,Y 261.246,Z 542.908,A -85,B 0,C 180,E1 -18993.085,E2 -18993.085} C_VEL
LIN {X 0,Y 265.242,Z 555.715,A -85,B 0,C 180,E1 -18994.82,E2 -18994.82} C_VEL
LIN {X 0,Y 268.397,Z 567.724,A -85,B 0,C 180,E1 -18996.579,E2 -18996.579} C_VEL
LIN {X 0,Y 269.461,Z 573.86,A -85,B 0,C 180,E1 -18997.494,E2 -18997.494} C_VEL
LIN {X 0,Y 266.786,Z 586.895,A -85,B 0,C 180,E1 -18999.095,E2 -18999.095} C_VEL
LIN {X 0,Y 263.933,Z 599.174,A -85,B 0,C 180,E1 -19000.937,E2 -19000.937} C_VEL
LIN {X 0,Y 260.878,Z 611.225,A -85,B 0,C 180,E1 -19003.148,E2 -19003.148} C_VEL
LIN {X 0,Y 258.102,Z 621.371,A -85,B 0,C 180,E1 -19005.396,E2 -19005.396} C_VEL
LIN {X 0,Y 255.356,Z 631.205,A -85,B 0,C 180,E1 -19008.037,E2 -19008.037} C_VEL
LIN {X 0,Y 252.97,Z 639.618,A -85,B 0,C 180,E1 -19010.793,E2 -19010.793} C_VEL
LIN {X 0,Y 250.856,Z 647.472,A -85,B 0,C 180,E1 -19013.969,E2 -19013.969} C_VEL
LIN {X 0,Y 249.438,Z 653.047,A -85,B 0,C 180,E1 -19016.796,E2 -19016.796} C_VEL
LIN {X 0,Y 248.402,Z 657.596,A -85,B 0,C 180,E1 -19019.677,E2 -19019.677} C_VEL
LIN {X 0,Y 247.623,Z 661.198,A -85,B 0,C 180,E1 -19022.633,E2 -19022.633} C_VEL
LIN {X 0,Y 247.188,Z 663.04,A -85,B 0,C 180,E1 -19024.655,E2 -19024.655} C_VEL
LIN {X 0,Y 246.891,Z 664.672,A -85,B 0,C 180,E1 -19027.15,E2 -19027.15} C_VEL
LIN {X 0,Y 246.825,Z 665.721,A -85,B 0,C 180,E1 -19029.754,E2 -19029.754} C_VEL
LIN {X 0,Y 247.017,Z 665.946,A -85,B 0,C 180,E1 -19033.066,E2 -19033.066} C_VEL
LIN {X 0,Y 247.301,Z 665.5,A -85,B 0,C 180,E1 -19035.273,E2 -19035.273} C_VEL
LIN {X 0,Y 247.793,Z 664.471,A -85,B 0,C 180,E1 -19037.512,E2 -19037.512} C_VEL
LIN {X 0,Y 248.503,Z 662.884,A -85,B 0,C 180,E1 -19039.782,E2 -19039.782} C_VEL
LIN {X 0,Y 249.82,Z 659.693,A -85,B 0,C 180,E1 -19042.983,E2 -19042.983} C_VEL
LIN {X 0,Y 251.598,Z 655.502,A -85,B 0,C 180,E1 -19046.035,E2 -19046.035} C_VEL
LIN {X 0,Y 253.972,Z 650.011,A -85,B 0,C 180,E1 -19049.075,E2 -19049.075} C_VEL
LIN {X 0,Y 257.155,Z 642.551,A -85,B 0,C 180,E1 -19052.314,E2 -19052.314} C_VEL
LIN {X 0,Y 260.685,Z 634.074,A -85,B 0,C 180,E1 -19055.216,E2 -19055.216} C_VEL
LIN {X 0,Y 264.37,Z 624.92,A -85,B 0,C 180,E1 -19057.739,E2 -19057.739} C_VEL
LIN {X 0,Y 268.225,Z 614.571,A -85,B 0,C 180,E1 -19060.084,E2 -19060.084} C_VEL
LIN {X 0,Y 272.367,Z 602.614,A -85,B 0,C 180,E1 -19062.292,E2 -19062.292} C_VEL
LIN {X 0,Y 276.157,Z 590.37,A -85,B 0,C 180,E1 -19064.124,E2 -19064.124} C_VEL
LIN {X 0,Y 278.337,Z 582.157,A -85,B 0,C 180,E1 -19065.183,E2 -19065.183} C_VEL
LIN {X 0,Y 276.541,Z 572.337,A -85,B 0,C 180,E1 -19067.151,E2 -19067.151} C_VEL
LIN {X 0,Y 273.693,Z 562.31,A -85,B 0,C 180,E1 -19069.27,E2 -19069.27} C_VEL
LIN {X 0,Y 270.783,Z 554.466,A -85,B 0,C 180,E1 -19071.04,E2 -19071.04} C_VEL
LIN {X 0,Y 266.345,Z 545.089,A -85,B 0,C 180,E1 -19073.405,E2 -19073.405} C_VEL
LIN {X 0,Y 263.48,Z 540.415,A -85,B 0,C 180,E1 -19074.806,E2 -19074.806} C_VEL
LIN {X 0,Y 260.93,Z 536.394,A -85,B 0,C 180,E1 -19076.096,E2 -19076.096} C_VEL
LIN {X 0,Y 258.536,Z 533.128,A -85,B 0,C 180,E1 -19077.273,E2 -19077.273} C_VEL
LIN {X 0,Y 257.657,Z 531.586,A -85,B 0,C 180,E1 -19077.752,E2 -19077.752} C_VEL
LIN {X 0,Y 255.52,Z 528.972,A -85,B 0,C 180,E1 -19078.867,E2 -19078.867} C_VEL
LIN {X 0,Y 254.252,Z 526.641,A -85,B 0,C 180,E1 -19079.603,E2 -19079.603} C_VEL
LIN {X 0,Y 251.575,Z 524.356,A -85,B 0,C 180,E1 -19080.999,E2 -19080.999} C_VEL
LIN {X 0,Y 250.232,Z 521.745,A -85,B 0,C 180,E1 -19081.911,E2 -19081.911} C_VEL
LIN {X 0,Y 250.148,Z 521.403,A -85,B 0,C 180,E1 -19082.012,E2 -19082.012} C_VEL
LIN {X 0,Y 249.947,Z 521.109,A -85,B 0,C 180,E1 -19086.457,E2 -19086.457} C_VEL
LIN {X 0,Y 249.914,Z 521.148,A -85,B 0,C 180,E1 -19090.181,E2 -19090.181} C_VEL
LIN {X 0,Y 249.842,Z 521.622,A -85,B 0,C 180,E1 -19094.664,E2 -19094.664} C_VEL
LIN {X 0,Y 249.892,Z 522.256,A -85,B 0,C 180,E1 -19098.02,E2 -19098.02} C_VEL
LIN {X 0,Y 249.901,Z 522.537,A -85,B 0,C 180,E1 -19099.159,E2 -19099.159} C_VEL
LIN {X 0,Y 249.317,Z 523.05,A -85,B 0,C 180,E1 -19100.501,E2 -19100.501} C_VEL
LIN {X 0,Y 246.624,Z 524.385,A -85,B 0,C 180,E1 -19102.684,E2 -19102.684} C_VEL
LIN {X 0,Y 244.348,Z 525.581,A -85,B 0,C 180,E1 -19104.458,E2 -19104.458} C_VEL
LIN {X 0,Y 243.431,Z 526.356,A -85,B 0,C 180,E1 -19105.834,E2 -19105.834} C_VEL
LIN {X 0,Y 243.39,Z 526.569,A -85,B 0,C 180,E1 -19106.3,E2 -19106.3} C_VEL
LIN {X 0,Y 243.657,Z 528.362,A -85,B 0,C 180,E1 -19110.082,E2 -19110.082} C_VEL
LIN {X 0,Y 244.092,Z 531.037,A -85,B 0,C 180,E1 -19114.655,E2 -19114.655} C_VEL
LIN {X 0,Y 245.262,Z 534.124,A -85,B 0,C 180,E1 -19115.656,E2 -19115.656} C_VEL
LIN {X 0,Y 247.607,Z 537.334,A -85,B 0,C 180,E1 -19117.235,E2 -19117.235} C_VEL
LIN {X 0,Y 248.851,Z 538.62,A -85,B 0,C 180,E1 -19117.983,E2 -19117.983} C_VEL
LIN {X 0,Y 250.491,Z 542.289,A -85,B 0,C 180,E1 -19119.067,E2 -19119.067} C_VEL
LIN {X 0,Y 252.833,Z 545.421,A -85,B 0,C 180,E1 -19120.392,E2 -19120.392} C_VEL
LIN {X 0,Y 254.701,Z 549.471,A -85,B 0,C 180,E1 -19121.528,E2 -19121.528} C_VEL
LIN {X 0,Y 256.119,Z 551.732,A -85,B 0,C 180,E1 -19122.275,E2 -19122.275} C_VEL
LIN {X 0,Y 258.282,Z 556.222,A -85,B 0,C 180,E1 -19123.521,E2 -19123.521} C_VEL
LIN {X 0,Y 260.462,Z 561.738,A -85,B 0,C 180,E1 -19124.823,E2 -19124.823} C_VEL
LIN {X 0,Y 263.216,Z 571.343,A -85,B 0,C 180,E1 -19126.788,E2 -19126.788} C_VEL
LIN {X 0,Y 265.616,Z 583.062,A -85,B 0,C 180,E1 -19128.944,E2 -19128.944} C_VEL
LIN {X 0,Y 266.892,Z 594.771,A -85,B 0,C 180,E1 -19130.997,E2 -19130.997} C_VEL
LIN {X 0,Y 267.175,Z 606.544,A -85,B 0,C 180,E1 -19133.019,E2 -19133.019} C_VEL
LIN {X 0,Y 266.339,Z 618.384,A -85,B 0,C 180,E1 -19135.087,E2 -19135.087} C_VEL
LIN {X 0,Y 262.029,Z 631.097,A -85,B 0,C 180,E1 -19137.102,E2 -19137.102} C_VEL
LIN {X 0,Y 257.855,Z 642.253,A -85,B 0,C 180,E1 -19139.266,E2 -19139.266} C_VEL
LIN {X 0,Y 253.501,Z 653.251,A -85,B 0,C 180,E1 -19141.881,E2 -19141.881} C_VEL
LIN {X 0,Y 250.044,Z 662.058,A -85,B 0,C 180,E1 -19144.455,E2 -19144.455} C_VEL
LIN {X 0,Y 247.23,Z 669.284,A -85,B 0,C 180,E1 -19146.991,E2 -19146.991} C_VEL
LIN {X 0,Y 244.698,Z 676.032,A -85,B 0,C 180,E1 -19149.839,E2 -19149.839} C_VEL
LIN {X 0,Y 242.422,Z 682.311,A -85,B 0,C 180,E1 -19153.147,E2 -19153.147} C_VEL
LIN {X 0,Y 241.009,Z 687.241,A -85,B 0,C 180,E1 -19156.509,E2 -19156.509} C_VEL
LIN {X 0,Y 240.177,Z 690.911,A -85,B 0,C 180,E1 -19159.887,E2 -19159.887} C_VEL
LIN {X 0,Y 239.953,Z 693.397,A -85,B 0,C 180,E1 -19163.271,E2 -19163.271} C_VEL
LIN {X 0,Y 240.025,Z 694.724,A -85,B 0,C 180,E1 -19166.642,E2 -19166.642} C_VEL
LIN {X 0,Y 240.186,Z 694.871,A -85,B 0,C 180,E1 -19169.999,E2 -19169.999} C_VEL
LIN {X 0,Y 240.1,Z 693.745,A -85,B 0,C 180,E1 -19173.355,E2 -19173.355} C_VEL
LIN {X 0,Y 240.09,Z 692.358,A -85,B 0,C 180,E1 -19175.587,E2 -19175.587} C_VEL
LIN {X 0,Y 240.084,Z 689.732,A -85,B 0,C 180,E1 -19178.415,E2 -19178.415} C_VEL
LIN {X 0,Y 240.504,Z 685.428,A -85,B 0,C 180,E1 -19181.802,E2 -19181.802} C_VEL
LIN {X 0,Y 241.545,Z 679.711,A -85,B 0,C 180,E1 -19185.18,E2 -19185.18} C_VEL
LIN {X 0,Y 243.258,Z 672.432,A -85,B 0,C 180,E1 -19188.529,E2 -19188.529} C_VEL
LIN {X 0,Y 245.3,Z 664.622,A -85,B 0,C 180,E1 -19191.424,E2 -19191.424} C_VEL
LIN {X 0,Y 248.053,Z 655.242,A -85,B 0,C 180,E1 -19194.255,E2 -19194.255} C_VEL
LIN {X 0,Y 250.638,Z 645.678,A -85,B 0,C 180,E1 -19196.655,E2 -19196.655} C_VEL
LIN {X 0,Y 253.793,Z 634.365,A -85,B 0,C 180,E1 -19198.985,E2 -19198.985} C_VEL
LIN {X 0,Y 257.097,Z 621.998,A -85,B 0,C 180,E1 -19201.061,E2 -19201.061} C_VEL
LIN {X 0,Y 259.027,Z 613.286,A -85,B 0,C 180,E1 -19202.301,E2 -19202.301} C_VEL
LIN {X 0,Y 258.27,Z 600.018,A -85,B 0,C 180,E1 -19204.291,E2 -19204.291} C_VEL
LIN {X 0,Y 256.675,Z 587.041,A -85,B 0,C 180,E1 -19206.048,E2 -19206.048} C_VEL
LIN {X 0,Y 253.91,Z 571.636,A -85,B 0,C 180,E1 -19207.921,E2 -19207.921} C_VEL
LIN {X 0,Y 250.212,Z 556.667,A -85,B 0,C 180,E1 -19209.593,E2 -19209.593} C_VEL
LIN {X 0,Y 245.696,Z 542.401,A -85,B 0,C 180,E1 -19211.064,E2 -19211.064} C_VEL
LIN {X 0,Y 244.684,Z 539.428,A -85,B 0,C 180,E1 -19211.359,E2 -19211.359} C_VEL
LIN {X 0,Y 244.602,Z 538.628,A -85,B 0,C 180,E1 -19211.431,E2 -19211.431} C_VEL
LIN {X 0,Y 244.933,Z 535.614,A -85,B 0,C 180,E1 -19214.166,E2 -19214.166} C_VEL
LIN {X 0,Y 244.363,Z 532.195,A -85,B 0,C 180,E1 -19217.48,E2 -19217.48} C_VEL
LIN {X 0,Y 243.597,Z 528.594,A -85,B 0,C 180,E1 -19221.164,E2 -19221.164} C_VEL
LIN {X 0,Y 243.061,Z 525.371,A -85,B 0,C 180,E1 -19224.67,E2 -19224.67} C_VEL
LIN {X 0,Y 242.519,Z 521.962,A -85,B 0,C 180,E1 -19228.559,E2 -19228.559} C_VEL
LIN {X 0,Y 242.047,Z 518.96,A -85,B 0,C 180,E1 -19232.318,E2 -19232.318} C_VEL
LIN {X 0,Y 242.034,Z 518.963,A -85,B 0,C 180,E1 -19236.014,E2 -19236.014} C_VEL
LIN {X 0,Y 242.028,Z 518.966,A -85,B 0,C 180,E1 -19239.608,E2 -19239.608} C_VEL
LIN {X 0,Y 242.156,Z 518.947,A -85,B 0,C 180,E1 -19243.278,E2 -19243.278} C_VEL
LIN {X 0,Y 242.179,Z 518.937,A -85,B 0,C 180,E1 -19248.28,E2 -19248.28} C_VEL
LIN {X 0,Y 242.42,Z 518.895,A -85,B 0,C 180,E1 -19251.666,E2 -19251.666} C_VEL
LIN {X 0,Y 242.256,Z 518.932,A -85,B 0,C 180,E1 -19255.008,E2 -19255.008} C_VEL
LIN {X 0,Y 242.632,Z 518.878,A -85,B 0,C 180,E1 -19258.341,E2 -19258.341} C_VEL
LIN {X 0,Y 242.63,Z 518.865,A -85,B 0,C 180,E1 -19261.661,E2 -19261.661} C_VEL
LIN {X 0,Y 242.417,Z 518.912,A -85,B 0,C 180,E1 -19266.675,E2 -19266.675} C_VEL
LIN {X 0,Y 242.261,Z 518.918,A -85,B 0,C 180,E1 -19270.025,E2 -19270.025} C_VEL
LIN {X 0,Y 242.157,Z 518.935,A -85,B 0,C 180,E1 -19275.142,E2 -19275.142} C_VEL
LIN {X 0,Y 242.067,Z 518.955,A -85,B 0,C 180,E1 -19278.625,E2 -19278.625} C_VEL
LIN {X 0,Y 242.007,Z 518.947,A -85,B 0,C 180,E1 -19282.181,E2 -19282.181} C_VEL
LIN {X 0,Y 242.062,Z 518.94,A -85,B 0,C 180,E1 -19285.839,E2 -19285.839} C_VEL
LIN {X 0,Y 242.025,Z 518.964,A -85,B 0,C 180,E1 -19289.582,E2 -19289.582} C_VEL
LIN {X 0,Y 241.988,Z 518.953,A -85,B 0,C 180,E1 -19293.492,E2 -19293.492} C_VEL
LIN {X 0,Y 242.01,Z 518.949,A -85,B 0,C 180,E1 -19297.579,E2 -19297.579} C_VEL
LIN {X 0,Y 242.035,Z 518.96,A -85,B 0,C 180,E1 -19301.903,E2 -19301.903} C_VEL
LIN {X 0,Y 242.018,Z 518.943,A -85,B 0,C 180,E1 -19306.551,E2 -19306.551} C_VEL
LIN {X 0,Y 242.009,Z 518.966,A -85,B 0,C 180,E1 -19310.293,E2 -19310.293} C_VEL
LIN {X 0,Y 242.037,Z 518.951,A -85,B 0,C 180,E1 -19314.499,E2 -19314.499} C_VEL
LIN {X 0,Y 241.977,Z 518.969,A -85,B 0,C 180,E1 -19318.482,E2 -19318.482} C_VEL
LIN {X 0,Y 242.011,Z 518.958,A -85,B 0,C 180,E1 -19322.315,E2 -19322.315} C_VEL
LIN {X 0,Y 242.063,Z 518.959,A -85,B 0,C 180,E1 -19326.018,E2 -19326.018} C_VEL
LIN {X 0,Y 242.04,Z 518.951,A -85,B 0,C 180,E1 -19329.609,E2 -19329.609} C_VEL
LIN {X 0,Y 242.166,Z 518.946,A -85,B 0,C 180,E1 -19333.28,E2 -19333.28} C_VEL
LIN {X 0,Y 242.185,Z 518.943,A -85,B 0,C 180,E1 -19338.281,E2 -19338.281} C_VEL
LIN {X 0,Y 242.398,Z 518.914,A -85,B 0,C 180,E1 -19341.666,E2 -19341.666} C_VEL
LIN {X 0,Y 242.261,Z 518.928,A -85,B 0,C 180,E1 -19345.008,E2 -19345.008} C_VEL
LIN {X 0,Y 242.659,Z 518.941,A -85,B 0,C 180,E1 -19348.621,E2 -19348.621} C_VEL
LIN {X 0,Y 243.625,Z 521.716,A -85,B 0,C 180,E1 -19348.924,E2 -19348.924} C_VEL
LIN {X 0,Y 244.987,Z 523.852,A -85,B 0,C 180,E1 -19349.267,E2 -19349.267} C_VEL
LIN {X 0,Y 249.735,Z 533.579,A -85,B 0,C 180,E1 -19350.659,E2 -19350.659} C_VEL
LIN {X 0,Y 255.494,Z 546.385,A -85,B 0,C 180,E1 -19352.569,E2 -19352.569} C_VEL
LIN {X 0,Y 259.421,Z 559.444,A -85,B 0,C 180,E1 -19354.442,E2 -19354.442} C_VEL
LIN {X 0,Y 262.414,Z 571.767,A -85,B 0,C 180,E1 -19356.344,E2 -19356.344} C_VEL
